(* Logix 5000 project; controller ARS14002_PLC vendor 1 type 14 code 218 rev 30.11; software revision 30.01 *)

TASK MainTask (continuous, watchdog 500 ms) : MainProgram
TASK PeriodicTask (periodic, rate 100 ms, priority 5, watchdog 1500 ms) : MainProgPeriodic

MODULES
   Local : vendor 1 type 14 code 218 (5069 0, rev 30.11)
      MAIN_PROCESSOR_T3_ENET : 1756-ENBT (Ethernet 192.168.23.100, rev 6.1, Output RPI 10 ms)   // PWHMI TOWER 3 ETHERNET MODULE
         MAIN_PROCESSOR_T3 : vendor 1 type 14 code 92 (ICP 0, rev 24.1, $d5a89411$ RPI 500 ms)   // PWHMI TOWER 3 PROCESSOR
      ARS14002_VFD800A : vendor 1 type 142 code 2192 (Ethernet 192.168.201.20, rev 13.3, Output RPI 20 ms)   // Cryo Pump 800A
          : vendor 1 type 142 code 16544 (RhinoBP 5, rev 1.1)
          : vendor 1 type 142 code 32928 (RhinoBP 13, rev 1.1)
          : vendor 1 type 142 code 767 (RhinoBP 2, rev 2.5)
          : vendor 1 type 142 code 57760 (RhinoBP 6, rev 1.2)
          : vendor 1 type 142 code 416 (RhinoBP 4, rev 1.8)
          : vendor 1 type 142 code 33184 (RhinoBP 14, rev 2.5)
      ARS14002_VFD800B : vendor 1 type 142 code 2192 (Ethernet 192.168.201.21, rev 13.3, Output RPI 20 ms)   // Cryo Pump 800B
          : vendor 1 type 142 code 416 (RhinoBP 4, rev 1.8)
          : vendor 1 type 142 code 767 (RhinoBP 2, rev 2.5)
          : vendor 1 type 142 code 32928 (RhinoBP 13, rev 1.1)
          : vendor 1 type 142 code 57760 (RhinoBP 6, rev 1.2)
          : vendor 1 type 142 code 33184 (RhinoBP 14, rev 2.5)
          : vendor 1 type 142 code 16544 (RhinoBP 5, rev 1.1)
      ARS14002_FVNR550 : vendor 1 type 3 code 506 (Ethernet 192.168.201.25, rev 5.1, Output RPI 20 ms)   // Vent Stack FAN-550
      ARS14002_FVR800C : vendor 1 type 3 code 548 (Ethernet 192.168.201.22, rev 5.1, Output RPI 20 ms)   // Cryo Pump 800C
      ARS14002_FVR800D : vendor 1 type 3 code 548 (Ethernet 192.168.201.23, rev 5.1, Output RPI 20 ms)   // Cryo Pump 800D
      MCP_S5 : 5069-IF8 (5069 5, rev 2.1, StandardDataDriven RPI 100 ms)
      MCP_S1 : 5069-IB16 (5069 1, rev 2.1, StandardDataDriven RPI 5 ms)
      MCP_S3 : vendor 1 type 7 code 1213 (5069 3, rev 3.1, StandardDataDriven RPI 5 ms)
      MCP_S4 : vendor 1 type 7 code 1213 (5069 4, rev 3.1, StandardDataDriven RPI 5 ms)
      MCP_S2 : vendor 1 type 7 code 1213 (5069 2, rev 3.1, StandardDataDriven RPI 5 ms)
      ARS14002_RCP1000 : 1734-AENTR (Ethernet 192.168.201.6, rev 5.1, Output RPI 20 ms)
         RCP1000_S13 : vendor 1 type 115 code 210 (PointIO 13, rev 3.1, Input RPI 80 ms)
         RCP1000_S1 : 1734-IB8 (PointIO 1, rev 3.1)
         RCP1000_S8 : vendor 1 type 115 code 49 (PointIO 8, rev 3.1, Input RPI 80 ms)
         RCP1000_S10 : vendor 1 type 115 code 49 (PointIO 10, rev 3.1, Input RPI 80 ms)
         RCP1000_S11 : vendor 1 type 115 code 49 (PointIO 11, rev 3.1, Input RPI 80 ms)
         RCP1000_S12 : vendor 1 type 115 code 210 (PointIO 12, rev 3.1, Input RPI 80 ms)
         RCP1000_S7 : vendor 1 type 115 code 49 (PointIO 7, rev 3.1, Input RPI 80 ms)
         RCP1000_S17 : vendor 1 type 115 code 49 (PointIO 17, rev 3.1, Input RPI 80 ms)
         RCP1000_S18 : vendor 1 type 115 code 49 (PointIO 18, rev 3.1, Input RPI 80 ms)
         RCP1000_S9 : vendor 1 type 115 code 49 (PointIO 9, rev 3.1, Input RPI 80 ms)
         RCP1000_S14 : vendor 1 type 115 code 210 (PointIO 14, rev 3.1, Input RPI 80 ms)
         RCP1000_S2 : 1734-IB8 (PointIO 2, rev 3.1)
         RCP1000_S3 : 1734-IB8 (PointIO 3, rev 3.1)
         RCP1000_S15 : vendor 1 type 115 code 211 (PointIO 15, rev 3.1, Output RPI 80 ms)
         RCP1000_S4 : 1734-OB8 (PointIO 4, rev 3.1)
         RCP1000_S6 : 1734-OB8 (PointIO 6, rev 3.1)
         RCP1000_S5 : 1734-OB8 (PointIO 5, rev 3.1)
         RCP1000_S16 : vendor 1 type 115 code 211 (PointIO 16, rev 3.1, Output RPI 80 ms)
      ARS14002_RCP600 : 1734-AENTR (Ethernet 192.168.201.4, rev 5.1, Output RPI 20 ms)
         RCP600_S7 : vendor 1 type 115 code 49 (PointIO 7, rev 3.1, Input RPI 80 ms)
         RCP600_S1 : 1734-IB8 (PointIO 1, rev 3.1)
         RCP600_S11 : vendor 1 type 115 code 210 (PointIO 11, rev 3.1, Input RPI 80 ms)
         RCP600_S9 : vendor 1 type 115 code 210 (PointIO 9, rev 3.1, Input RPI 80 ms)
         RCP600_S6 : vendor 1 type 115 code 49 (PointIO 6, rev 3.1, Input RPI 80 ms)
         RCP600_S10 : vendor 1 type 115 code 210 (PointIO 10, rev 3.1, Input RPI 80 ms)
         RCP600_S8 : vendor 1 type 115 code 49 (PointIO 8, rev 3.1, Input RPI 80 ms)
         RCP600_S5 : vendor 1 type 115 code 49 (PointIO 5, rev 3.1, Input RPI 80 ms)
         RCP600_S4 : 1734-OB8 (PointIO 4, rev 3.1)
         RCP600_S3 : 1734-OB8 (PointIO 3, rev 3.1)
         RCP600_S12 : vendor 1 type 115 code 211 (PointIO 12, rev 3.1, Output RPI 80 ms)
         RCP600_S13 : vendor 1 type 115 code 211 (PointIO 13, rev 3.1, Output RPI 80 ms)
         RCP600_S2 : 1734-OB8 (PointIO 2, rev 3.1)
      ARS14002_RCP800 : 1734-AENTR (Ethernet 192.168.201.5, rev 5.1, Output RPI 20 ms)
         RCP800_S23 : vendor 1 type 115 code 210 (PointIO 23, rev 3.1, Input RPI 80 ms)
         RCP800_S21 : vendor 1 type 115 code 210 (PointIO 21, rev 3.1, Input RPI 80 ms)
         RCP800_S17 : 1734-IR2 (PointIO 17, rev 3.1, Input RPI 80 ms)
         RCP800_S13 : 1734-IR2 (PointIO 13, rev 3.1, Input RPI 80 ms)
         RCP800_S2 : 1734-IB8 (PointIO 2, rev 3.1)
         RCP800_S16 : 1734-IR2 (PointIO 16, rev 3.1, Input RPI 80 ms)
         RCP800_S12 : vendor 1 type 115 code 49 (PointIO 12, rev 3.1, Input RPI 80 ms)
         RCP800_S22 : vendor 1 type 115 code 210 (PointIO 22, rev 3.1, Input RPI 80 ms)
         RCP800_S20 : 1734-IR2 (PointIO 20, rev 3.1, Input RPI 80 ms)
         RCP800_S24 : vendor 1 type 115 code 210 (PointIO 24, rev 3.1, Input RPI 80 ms)
         RCP800_S8 : 1734-IR2 (PointIO 8, rev 3.1, Input RPI 80 ms)
         RCP800_S11 : vendor 1 type 115 code 49 (PointIO 11, rev 3.1, Input RPI 80 ms)
         RCP800_S3 : 1734-IB8 (PointIO 3, rev 3.1)
         RCP800_S18 : 1734-IR2 (PointIO 18, rev 3.1, Input RPI 80 ms)
         RCP800_S14 : 1734-IR2 (PointIO 14, rev 3.1, Input RPI 80 ms)
         RCP800_S1 : 1734-IB8 (PointIO 1, rev 3.1)
         RCP800_S15 : 1734-IR2 (PointIO 15, rev 3.1, Input RPI 80 ms)
         RCP800_S10 : vendor 1 type 115 code 49 (PointIO 10, rev 3.1, Input RPI 80 ms)
         RCP800_S9 : 1734-IR2 (PointIO 9, rev 3.1, Input RPI 80 ms)
         RCP800_S19 : 1734-IR2 (PointIO 19, rev 3.1, Input RPI 80 ms)
         RCP800_S4 : 1734-OB8 (PointIO 4, rev 3.1)
         RCP800_S5 : 1734-OB8 (PointIO 5, rev 3.1)
         RCP800_S25 : vendor 1 type 115 code 211 (PointIO 25, rev 3.1, Output RPI 80 ms)
         RCP800_S7 : 1734-OB8 (PointIO 7, rev 3.1)
         RCP800_S6 : 1734-OB8 (PointIO 6, rev 3.1)
      ARS14002_RCP100 : 1734-AENTR (Ethernet 192.168.201.3, rev 5.1, Output RPI 20 ms)
         RCP100_S3 : vendor 1 type 115 code 49 (PointIO 3, rev 3.1, Input RPI 80 ms)
         RCP100_S5 : vendor 1 type 115 code 210 (PointIO 5, rev 3.1, Input RPI 80 ms)
         RCP100_S4 : vendor 1 type 115 code 49 (PointIO 4, rev 3.1, Input RPI 80 ms)
         RCP100_S6 : vendor 1 type 115 code 210 (PointIO 6, rev 3.1, Input RPI 80 ms)
         RCP100_S1 : 1734-IB8 (PointIO 1, rev 3.1)
         RCP100_S9 : 1734-OB8 (PointIO 9, rev 3.1)
         RCP100_S2 : 1734-OB8 (PointIO 2, rev 3.1)
         RCP100_S7 : vendor 1 type 115 code 211 (PointIO 7, rev 3.1, Output RPI 80 ms)
         RCP100_S8 : vendor 1 type 115 code 211 (PointIO 8, rev 3.1, Output RPI 80 ms)
END_MODULES

TYPE UDT_IPC :
STRUCT
   ConnectionStatus : CONNECTION_STATUS;
   BOOL : BOOL[32];
   REAL : REAL[32];
   DINT : DINT[32];
END_STRUCT
END_TYPE

ADD_ON_INSTRUCTION CM_AI_SCL   (* revision 2.0, vendor EVERWORKS *)
// Analog Input
VAR_INPUT
   RawMin : INT := 4000; {required}   // Config Raw Min
   RawMax : INT := 20000; {required}   // Config Raw Max
   EuMin : REAL; {visible}   // Config Min EU
   EuMax : REAL := 100.0; {visible}   // Config Max EU
   In_Raw : INT; {required}   // Channel Raw Count
END_VAR
VAR_OUTPUT
   Percent : REAL; {access Read Only}   // Scaled % of PV
   PV : REAL; {access Read Only, visible}   // Scaled PV
END_VAR

ROUTINE Logic   (* ladder *)
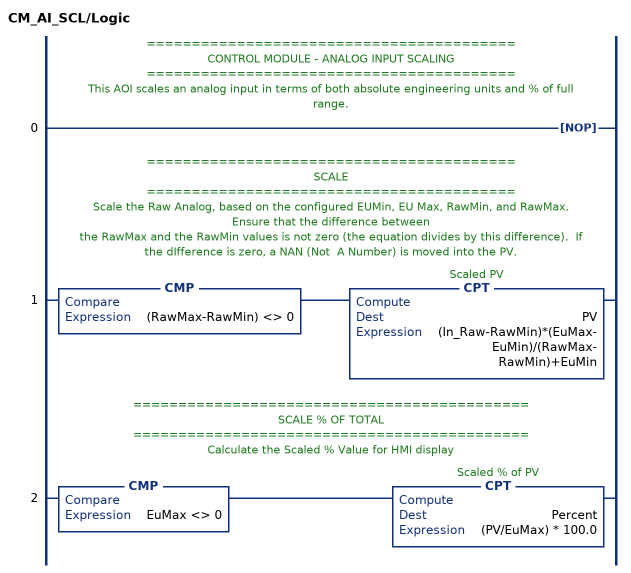
   // =========================================
   // CONTROL MODULE - ANALOG INPUT SCALING
   // =========================================
   // This AOI scales an analog input in terms of both absolute engineering units and % of full range.
   0: NOP();
   // =========================================
   // SCALE
   // =========================================
   // Scale the Raw Analog, based on the configured EUMin, EU Max, RawMin, and RawMax.  Ensure that the difference between
   // the RawMax and the RawMin values is not zero (the equation divides by this difference).  If the dIfference is zero, a NAN (Not  A Number) is moved into the PV.
   1: CMP((RawMax-RawMin) <> 0)CPT(PV,(In_Raw-RawMin)*(EuMax-EuMin)/(RawMax-RawMin)+EuMin);
   // ============================================
   // SCALE % OF TOTAL
   // ============================================
   // Calculate the Scaled % Value for HMI display
   2: CMP(EuMax <> 0)CPT(Percent,(PV/EuMax) * 100.0);
END_ROUTINE
END_ADD_ON_INSTRUCTION

ADD_ON_INSTRUCTION CM_AI_SCL_ALT   (* revision 2.0, vendor EVERWORKS *)
// Analog Input with Alt Scaling
VAR_INPUT
   RawMin : INT := 4000; {required}   // Config Raw Min
   RawMax : INT := 20000; {required}   // Config Raw Max
   EuMin : REAL; {visible}   // Config Min EU
   EuMax : REAL := 100.0; {visible}   // Config Max EU
   AltScaleMultiplier : REAL; {required}   // Alternate Scale Multiplier
   In_Raw : INT; {required}   // Channel Raw Count
END_VAR
VAR_OUTPUT
   Percent : REAL; {access Read Only}   // Scaled % of PV
   PV : REAL; {access Read Only, visible}   // Scaled PV
   AltScalePV : REAL; {visible}   // Alternate Scaled PV
END_VAR

ROUTINE Logic   (* ladder *)
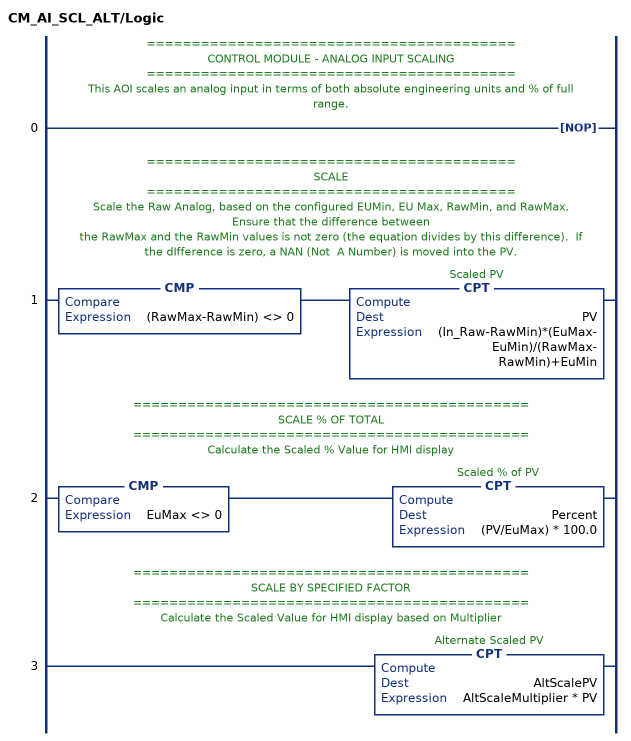
   // =========================================
   // CONTROL MODULE - ANALOG INPUT SCALING
   // =========================================
   // This AOI scales an analog input in terms of both absolute engineering units and % of full range.
   0: NOP();
   // =========================================
   // SCALE
   // =========================================
   // Scale the Raw Analog, based on the configured EUMin, EU Max, RawMin, and RawMax.  Ensure that the difference between
   // the RawMax and the RawMin values is not zero (the equation divides by this difference).  If the dIfference is zero, a NAN (Not  A Number) is moved into the PV.
   1: CMP((RawMax-RawMin) <> 0)CPT(PV,(In_Raw-RawMin)*(EuMax-EuMin)/(RawMax-RawMin)+EuMin);
   // ============================================
   // SCALE % OF TOTAL
   // ============================================
   // Calculate the Scaled % Value for HMI display
   2: CMP(EuMax <> 0)CPT(Percent,(PV/EuMax) * 100.0);
   // ============================================
   // SCALE BY SPECIFIED FACTOR
   // ============================================
   // Calculate the Scaled Value for HMI display based on Multiplier
   3: CPT(AltScalePV,AltScaleMultiplier * PV);
END_ROUTINE
END_ADD_ON_INSTRUCTION

ADD_ON_INSTRUCTION CM_AO_SCL   (* revision 2.0, vendor EVERWORKS *)
// Analog Output
VAR_OUTPUT
   EngValue : REAL; {access Read Only, visible}   // Scaled Engineering Value
   Percent : REAL; {access Read Only}   // Scaled % of PV
   Out_Raw : INT; {required}   // Channel Raw Count
END_VAR
VAR_INPUT
   EuMin : REAL; {visible}   // Config Min EU
   EuMax : REAL := 100.0; {visible}   // Config Max EU
   RawMin : INT := 4000; {required}   // Config Raw Min
   RawMax : INT := 20000; {required}   // Config Raw Max
END_VAR

ROUTINE Logic   (* ladder *)
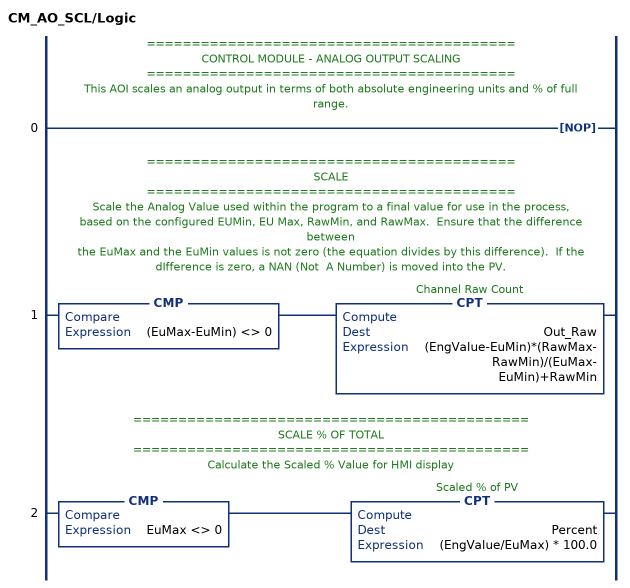
   // =========================================
   // CONTROL MODULE - ANALOG OUTPUT SCALING
   // =========================================
   // This AOI scales an analog output in terms of both absolute engineering units and % of full range.
   0: NOP();
   // =========================================
   // SCALE
   // =========================================
   // Scale the Analog Value used within the program to a final value for use in the process, based on the configured EUMin, EU Max, RawMin, and RawMax.  Ensure that the difference between
   // the EuMax and the EuMin values is not zero (the equation divides by this difference).  If the dIfference is zero, a NAN (Not  A Number) is moved into the PV.
   1: CMP((EuMax-EuMin) <> 0)CPT(Out_Raw,(EngValue-EuMin)*(RawMax-RawMin)/(EuMax-EuMin)+RawMin);
   // ============================================
   // SCALE % OF TOTAL
   // ============================================
   // Calculate the Scaled % Value for HMI display
   2: CMP(EuMax <> 0)CPT(Percent,(EngValue/EuMax) * 100.0);
END_ROUTINE
END_ADD_ON_INSTRUCTION

ADD_ON_INSTRUCTION CM_AO_VLV   (* revision 2.0, vendor EVERWORKS *)
// Modulating Valve
VAR_INPUT
   FailPos : BOOL; {required}   // Fail Position (0=Fail Closed, 1=Fail Open)
   EuMin : REAL; {visible}   // Config Min EU
   EuMax : REAL := 100.0; {visible}   // Config Max EU
   RawMin : INT := 4000; {required}   // Config Raw Min
   RawMax : INT := 20000; {required}   // Config Raw Max
   ZT : REAL; {required}   // Position Feedback (EU)
   EngValue : REAL; {access Read Only, visible}   // Scaled Engineering Value
END_VAR
VAR_OUTPUT
   Out_Raw : INT; {required}   // Channel Raw Count
   Alm_Dev : BOOL; {visible}   // Deviation Alarm
END_VAR
VAR_INPUT
   Alm_Dev_SP : REAL := 10.0;   // % Deviation between CV and ZT allowed
   Alm_Dev_TmrPre : DINT := 5;   // Deviation Alarm Delay Timer Preset (seconds)
END_VAR
VAR
   Alm_Dev_Tmr : TIMER := (PRE := 5000); {access None}   // Deviation Alarm Delay Timer
   Comp_Overshoot : REAL; {access None}   // ZT (position feedback) - CV (commanded position)
   Comp_Undershoot : REAL; {access None}   // CV (commanded position) - ZT (position feedback)
END_VAR

ROUTINE Logic   (* ladder *)
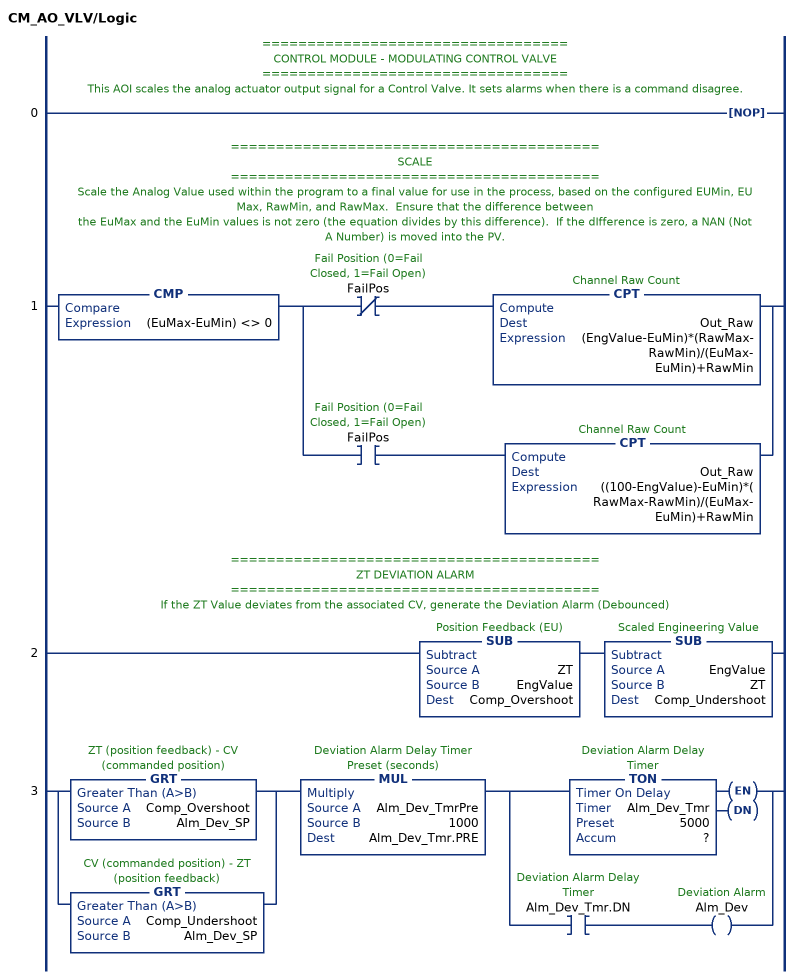
   // ==================================
   // CONTROL MODULE - MODULATING CONTROL VALVE
   // ==================================
   // This AOI scales the analog actuator output signal for a Control Valve. It sets alarms when there is a command disagree.
   0: NOP();
   // =========================================
   // SCALE
   // =========================================
   // Scale the Analog Value used within the program to a final value for use in the process, based on the configured EUMin, EU Max, RawMin, and RawMax.  Ensure that the difference between
   // the EuMax and the EuMin values is not zero (the equation divides by this difference).  If the dIfference is zero, a NAN (Not  A Number) is moved into the PV.
   1: CMP((EuMax-EuMin) <> 0)[XIO(FailPos) CPT(Out_Raw,(EngValue-EuMin)*(RawMax-RawMin)/(EuMax-EuMin)+RawMin) ,XIC(FailPos) CPT(Out_Raw,((100-EngValue)-EuMin)*(RawMax-RawMin)/(EuMax-EuMin)+RawMin) ];
   // =========================================
   // ZT DEVIATION ALARM
   // =========================================
   // If the ZT Value deviates from the associated CV, generate the Deviation Alarm (Debounced)
   2: SUB(ZT,EngValue,Comp_Overshoot)SUB(EngValue,ZT,Comp_Undershoot);
   3: [GRT(Comp_Overshoot,Alm_Dev_SP) ,GRT(Comp_Undershoot,Alm_Dev_SP) ]MUL(Alm_Dev_TmrPre,1000,Alm_Dev_Tmr.PRE)[TON(Alm_Dev_Tmr,?,?) ,XIC(Alm_Dev_Tmr.DN) OTE(Alm_Dev) ];
END_ROUTINE
END_ADD_ON_INSTRUCTION

ADD_ON_INSTRUCTION CM_DO_FVNR   (* revision 2.0, vendor EVERWORKS *)
// FVNR Starter
VAR_INPUT
   ILW : DINT;   // InterLocks Word
   Auto : BOOL; {visible}   // Starter Mode (0=Manual, 1=Auto)
   AlmCurrentLow_SP : REAL; {visible}   // Low Current Setpoint
   AlmCurrentHigh_SP : REAL := 999.0; {visible}   // High Current Setpoint
   Current : REAL; {access Read Only, visible}   // Motor Current Feedback
   Flt : BOOL; {visible}   // Fault Status
   AlmCD_TmrPre : DINT := 5;   // Command Disagree Alarm Delay Timer Preset (Seconds)
END_VAR
VAR_OUTPUT
   Intlk : BOOL; {access Read Only, visible}   // Interlocked Status
END_VAR
VAR_INPUT
   ProgStartReq : BOOL;   // Program Start Request
END_VAR
VAR_OUTPUT
   AlmCD : BOOL; {access Read Only, visible}   // Command Disagree Alarm
END_VAR
VAR_INPUT
   Running : BOOL; {visible}   // Motor Running Status
END_VAR
VAR_OUTPUT
   Out : BOOL; {required}   // Start Command
   AlmCurrentLow : BOOL; {visible}   // Low Current Alarm
   AlmCurrentHigh : BOOL; {visible}   // High Current Alarm
END_VAR
VAR_INPUT
   AlmCurrent_TmrPre : DINT := 5;   // Low Current Alarm Delay Timer Preset (Seconds)
   OperStartReq : BOOL;   // Manual Start Request
END_VAR
VAR
   AlmCD_Tmr : TIMER := (PRE := 5000); {access None}   // Command Disagree Alarm Delay Timer
   ILW_Desc : STRING[14];
   AlmCurrentLow_Tmr : TIMER := (PRE := 5000); {access None}   // Low Current Alarm Delay Timer
   AutoManTransOSR_SB : BOOL; {access None}
   AutoManTransOSR_OB : BOOL; {access None}
   AlmCurrentHigh_Tmr : TIMER := (PRE := 5000); {access None}   // High Current Alarm Delay Timer
END_VAR

ROUTINE Logic   (* ladder *)
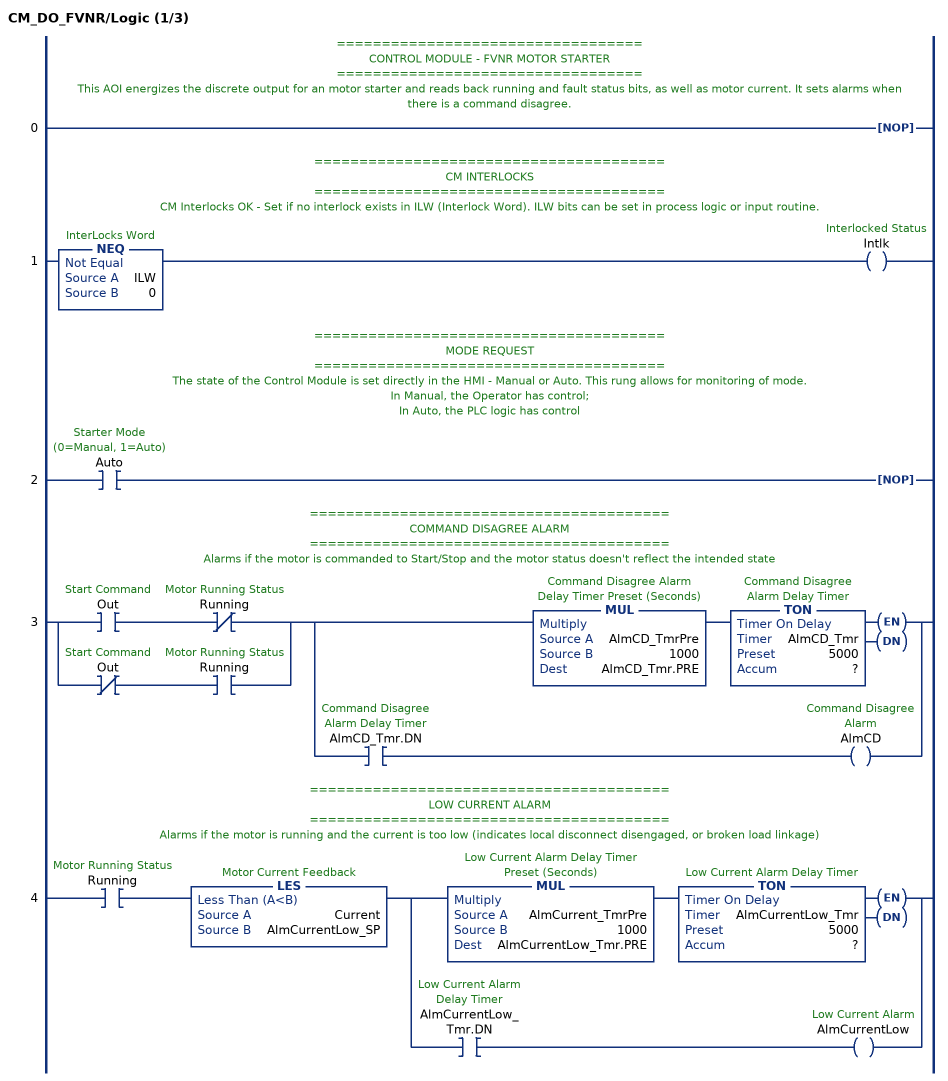
   // ==================================
   // CONTROL MODULE - FVNR MOTOR STARTER
   // ==================================
   // This AOI energizes the discrete output for an motor starter and reads back running and fault status bits, as well as motor current. It sets alarms when there is a command disagree.
   0: NOP();
   // =======================================
   // CM INTERLOCKS
   // =======================================
   // CM Interlocks OK - Set if no interlock exists in ILW (Interlock Word). ILW bits can be set in process logic or input routine.
   1: NEQ(ILW,0)OTE(Intlk);
   // =======================================
   // MODE REQUEST
   // =======================================
   // The state of the Control Module is set directly in the HMI - Manual or Auto. This rung allows for monitoring of mode.
   // In Manual, the Operator has control;
   //  In Auto, the PLC logic has control
   2: XIC(Auto)NOP();
   // ========================================
   // COMMAND DISAGREE ALARM
   // ========================================
   // Alarms if the motor is commanded to Start/Stop and the motor status doesn't reflect the intended state
   3: [XIC(Out) XIO(Running) ,XIO(Out) XIC(Running) ][MUL(AlmCD_TmrPre,1000,AlmCD_Tmr.PRE) TON(AlmCD_Tmr,?,?) ,XIC(AlmCD_Tmr.DN) OTE(AlmCD) ];
   // ========================================
   // LOW CURRENT ALARM
   // ========================================
   // Alarms if the motor is running and the current is too low (indicates local disconnect disengaged, or broken load linkage)
   4: XIC(Running)LES(Current,AlmCurrentLow_SP)[MUL(AlmCurrent_TmrPre,1000,AlmCurrentLow_Tmr.PRE) TON(AlmCurrentLow_Tmr,?,?) ,XIC(AlmCurrentLow_Tmr.DN) OTE(AlmCurrentLow) ];
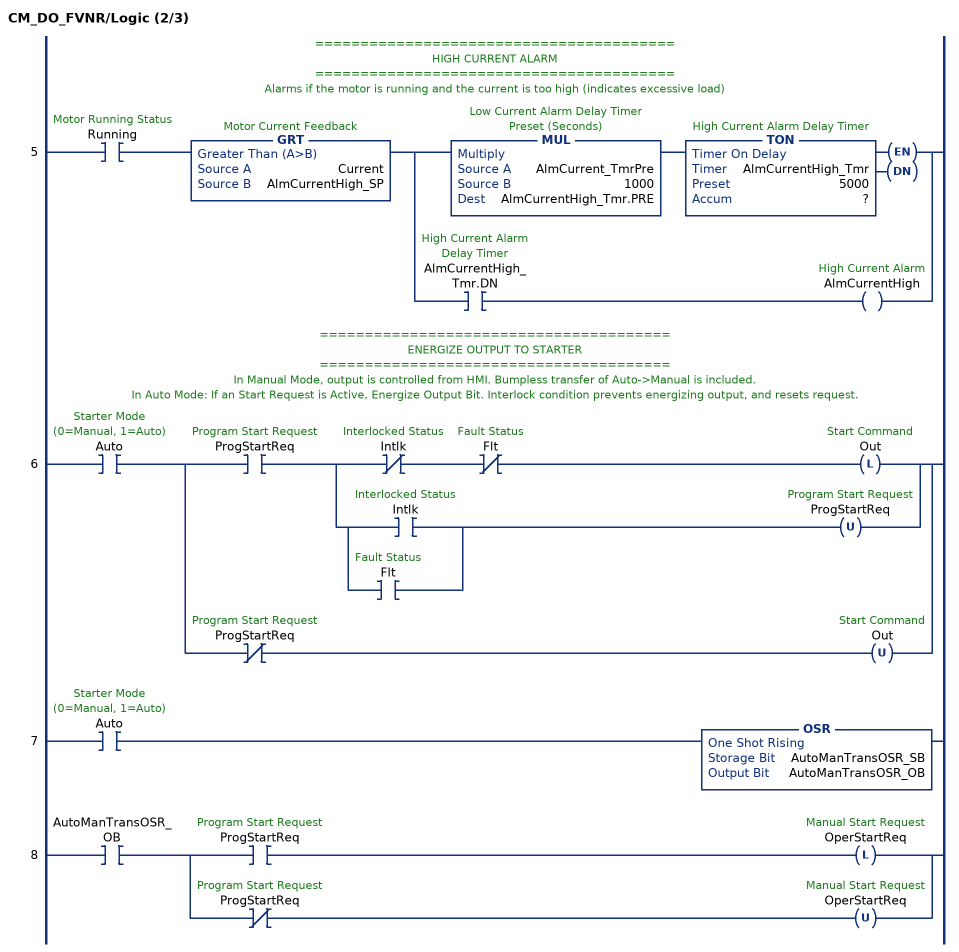
   // ========================================
   // HIGH CURRENT ALARM
   // ========================================
   // Alarms if the motor is running and the current is too high (indicates excessive load)
   5: XIC(Running)GRT(Current,AlmCurrentHigh_SP)[MUL(AlmCurrent_TmrPre,1000,AlmCurrentHigh_Tmr.PRE) TON(AlmCurrentHigh_Tmr,?,?) ,XIC(AlmCurrentHigh_Tmr.DN) OTE(AlmCurrentHigh) ];
   // =======================================
   // ENERGIZE OUTPUT TO STARTER
   // =======================================
   // In Manual Mode, output is controlled from HMI. Bumpless transfer of Auto->Manual is included.
   // In Auto Mode: If an Start Request is Active, Energize Output Bit. Interlock condition prevents energizing output, and resets request.
   6: XIC(Auto)[XIC(ProgStartReq) [XIO(Intlk) XIO(Flt) OTL(Out) ,[XIC(Intlk) ,XIC(Flt) ] OTU(ProgStartReq) ] ,XIO(ProgStartReq) OTU(Out) ];
   7: XIC(Auto)OSR(AutoManTransOSR_SB,AutoManTransOSR_OB);
   8: XIC(AutoManTransOSR_OB)[XIC(ProgStartReq) OTL(OperStartReq) ,XIO(ProgStartReq) OTU(OperStartReq) ];
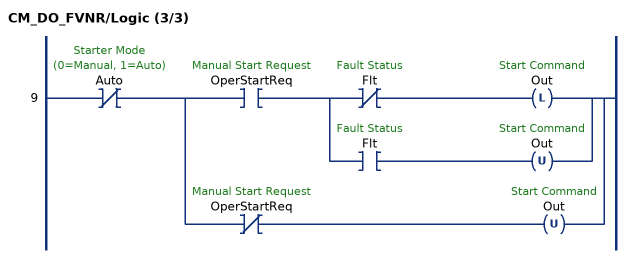
   9: XIO(Auto)[XIC(OperStartReq) [XIO(Flt) OTL(Out) ,XIC(Flt) OTU(Out) ] ,XIO(OperStartReq) OTU(Out) ];
END_ROUTINE
END_ADD_ON_INSTRUCTION

ADD_ON_INSTRUCTION CM_DO_FVR   (* revision 2.0, vendor EVERWORKS *)
// FVR Starter
VAR_INPUT
   ILW : DINT;   // InterLocks Word
   Auto : BOOL; {visible}   // Starter Mode (0=Manual, 1=Auto)
   AlmCurrentLow_SP : REAL; {visible}   // Low Current Setpoint
   AlmCurrentHigh_SP : REAL := 999.0; {visible}   // High Current Setpoint
   Current : REAL; {access Read Only, visible}   // Motor Current Feedback
   Flt : BOOL; {visible}   // Fault Status
   AlmCD_TmrPre : DINT := 5;   // Command Disagree Alarm Delay Timer Preset (Seconds)
END_VAR
VAR_OUTPUT
   Intlk : BOOL; {access Read Only, visible}   // Interlocked Status
END_VAR
VAR_INPUT
   ProgStartReq : BOOL;   // Program Start Request
END_VAR
VAR_OUTPUT
   AlmCD : BOOL; {access Read Only, visible}   // Command Disagree Alarm
END_VAR
VAR_INPUT
   Direction : BOOL; {visible}   // Motor Direction 0=Forward 1=Reverse
   RunningFwd : BOOL; {visible}   // Motor Running Forward Status
   RunningRvs : BOOL; {visible}   // Motor Running Reverse Status
END_VAR
VAR_OUTPUT
   OutFwd : BOOL; {required}   // Start Command Forward
   OutRvs : BOOL; {access Read Only, required}   // Start Command Reverse
   AlmCurrentLow : BOOL; {visible}   // Low Current Alarm
   AlmCurrentHigh : BOOL; {visible}   // High Current Alarm
END_VAR
VAR_INPUT
   AlmCurrent_TmrPre : DINT := 5;   // Low Current Alarm Delay Timer Preset (Seconds)
   OperStartReq : BOOL;   // Manual Start Request
END_VAR
VAR
   AlmCD_Tmr : TIMER := (PRE := 5000); {access None}   // Command Disagree Alarm Delay Timer
   ILW_Desc : STRING[14];
   AlmCurrentLow_Tmr : TIMER := (PRE := 5000); {access None}   // Low Current Alarm Delay Timer
   AutoManTransOSR_SB : BOOL; {access None}
   AutoManTransOSR_OB : BOOL; {access None}
   AlmCurrentHigh_Tmr : TIMER := (PRE := 5000); {access None}   // High Current Alarm Delay Timer
END_VAR

ROUTINE Logic   (* ladder *)
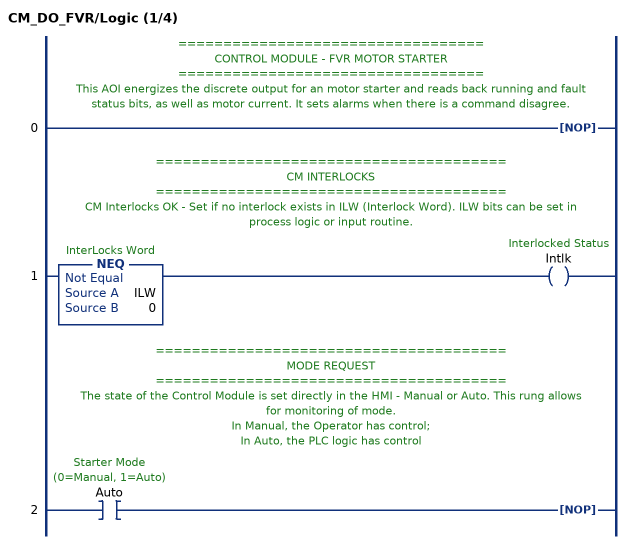
   // ==================================
   // CONTROL MODULE - FVR MOTOR STARTER
   // ==================================
   // This AOI energizes the discrete output for an motor starter and reads back running and fault status bits, as well as motor current. It sets alarms when there is a command disagree.
   0: NOP();
   // =======================================
   // CM INTERLOCKS
   // =======================================
   // CM Interlocks OK - Set if no interlock exists in ILW (Interlock Word). ILW bits can be set in process logic or input routine.
   1: NEQ(ILW,0)OTE(Intlk);
   // =======================================
   // MODE REQUEST
   // =======================================
   // The state of the Control Module is set directly in the HMI - Manual or Auto. This rung allows for monitoring of mode.
   // In Manual, the Operator has control;
   //  In Auto, the PLC logic has control
   2: XIC(Auto)NOP();
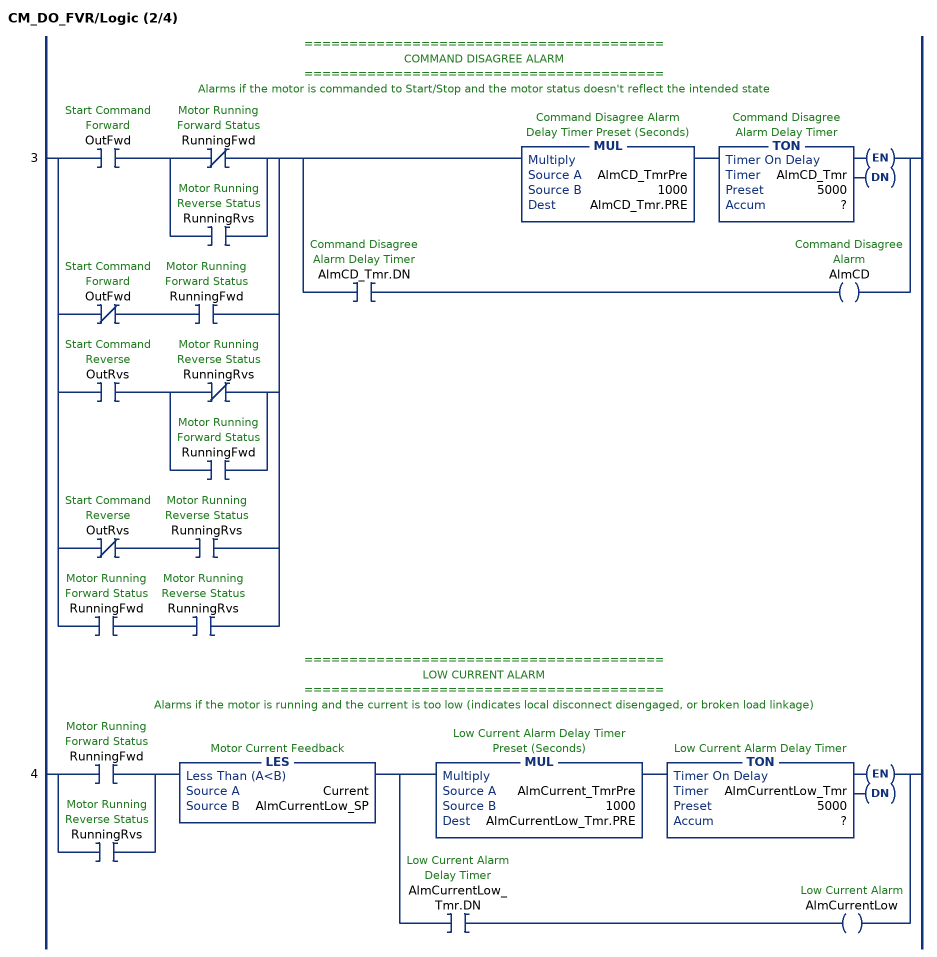
   // ========================================
   // COMMAND DISAGREE ALARM
   // ========================================
   // Alarms if the motor is commanded to Start/Stop and the motor status doesn't reflect the intended state
   3: [XIC(OutFwd) [XIO(RunningFwd) ,XIC(RunningRvs) ] ,XIO(OutFwd) XIC(RunningFwd) ,XIC(OutRvs) [XIO(RunningRvs) ,XIC(RunningFwd) ] ,XIO(OutRvs) XIC(RunningRvs) ,XIC(RunningFwd) XIC(RunningRvs) ][MUL(AlmCD_TmrPre,1000,AlmCD_Tmr.PRE) TON(AlmCD_Tmr,?,?) ,XIC(AlmCD_Tmr.DN) OTE(AlmCD) ];
   // ========================================
   // LOW CURRENT ALARM
   // ========================================
   // Alarms if the motor is running and the current is too low (indicates local disconnect disengaged, or broken load linkage)
   4: [XIC(RunningFwd) ,XIC(RunningRvs) ]LES(Current,AlmCurrentLow_SP)[MUL(AlmCurrent_TmrPre,1000,AlmCurrentLow_Tmr.PRE) TON(AlmCurrentLow_Tmr,?,?) ,XIC(AlmCurrentLow_Tmr.DN) OTE(AlmCurrentLow) ];
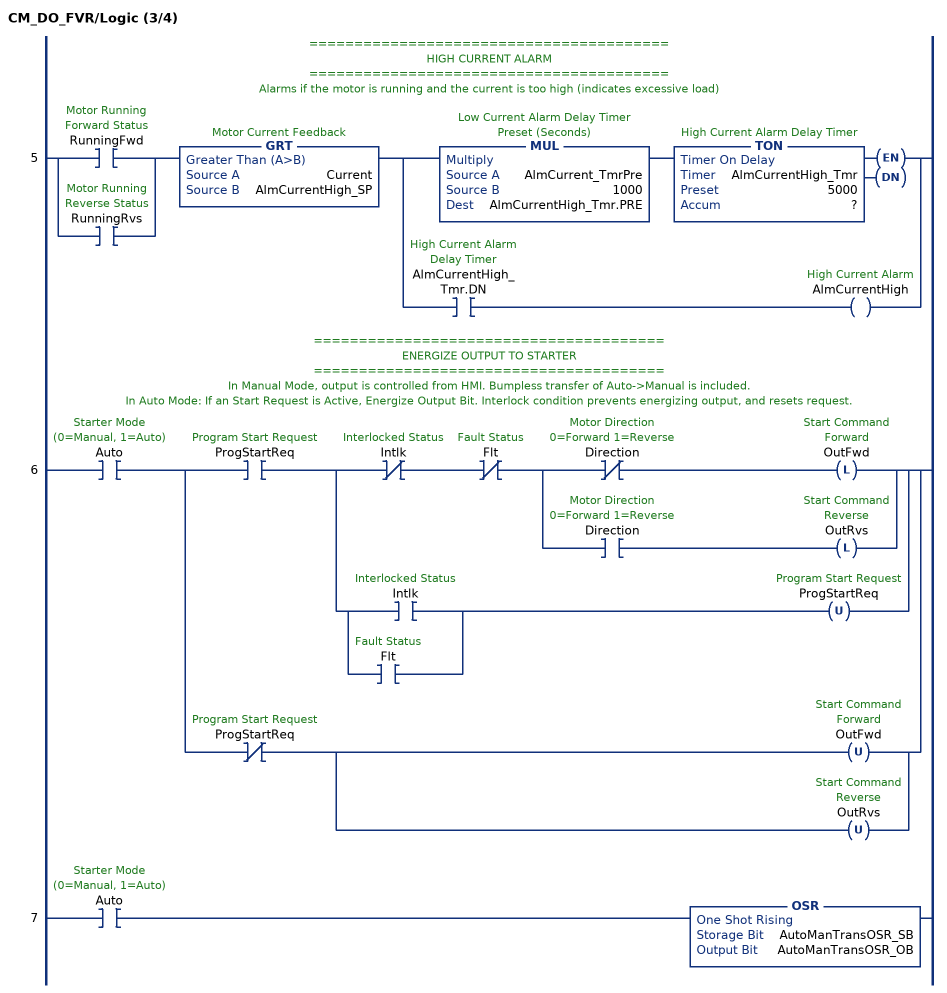
   // ========================================
   // HIGH CURRENT ALARM
   // ========================================
   // Alarms if the motor is running and the current is too high (indicates excessive load)
   5: [XIC(RunningFwd) ,XIC(RunningRvs) ]GRT(Current,AlmCurrentHigh_SP)[MUL(AlmCurrent_TmrPre,1000,AlmCurrentHigh_Tmr.PRE) TON(AlmCurrentHigh_Tmr,?,?) ,XIC(AlmCurrentHigh_Tmr.DN) OTE(AlmCurrentHigh) ];
   // =======================================
   // ENERGIZE OUTPUT TO STARTER
   // =======================================
   // In Manual Mode, output is controlled from HMI. Bumpless transfer of Auto->Manual is included.
   // In Auto Mode: If an Start Request is Active, Energize Output Bit. Interlock condition prevents energizing output, and resets request.
   6: XIC(Auto)[XIC(ProgStartReq) [XIO(Intlk) XIO(Flt) [XIO(Direction) OTL(OutFwd) ,XIC(Direction) OTL(OutRvs) ] ,[XIC(Intlk) ,XIC(Flt) ] OTU(ProgStartReq) ] ,XIO(ProgStartReq) [OTU(OutFwd) ,OTU(OutRvs) ] ];
   7: XIC(Auto)OSR(AutoManTransOSR_SB,AutoManTransOSR_OB);
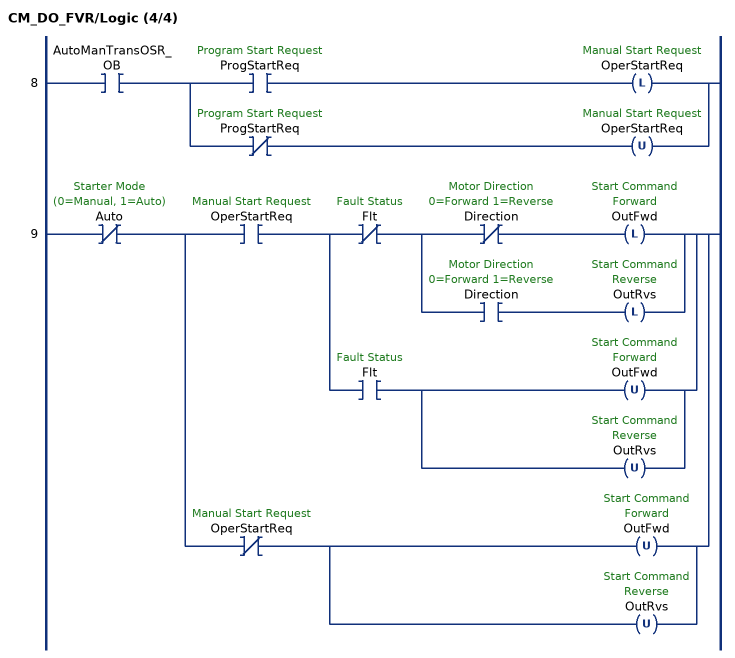
   8: XIC(AutoManTransOSR_OB)[XIC(ProgStartReq) OTL(OperStartReq) ,XIO(ProgStartReq) OTU(OperStartReq) ];
   9: XIO(Auto)[XIC(OperStartReq) [XIO(Flt) [XIO(Direction) OTL(OutFwd) ,XIC(Direction) OTL(OutRvs) ] ,XIC(Flt) [OTU(OutFwd) ,OTU(OutRvs) ] ] ,XIO(OperStartReq) [OTU(OutFwd) ,OTU(OutRvs) ] ];
END_ROUTINE
END_ADD_ON_INSTRUCTION

ADD_ON_INSTRUCTION CM_DO_GENERIC   (* revision 2.0, vendor EVERWORKS *)
// On/Off Device (No Feedback)
VAR_INPUT
   ILW : DINT;   // InterLocks Word
   FailPos : BOOL; {visible}   // Fail Position (0=Fail Closed, 1=Fail Open)
   Auto : BOOL; {visible}   // Device Mode (0=Manual, 1=Auto)
END_VAR
VAR_OUTPUT
   Intlk : BOOL; {access Read Only, visible}   // Interlocked Status
END_VAR
VAR_INPUT
   EnergizeReq : BOOL; {visible}   // Program Energize Request
END_VAR
VAR_OUTPUT
   Out : BOOL; {required}   // Energize Command
END_VAR
VAR_INPUT
   DeenergizeONS : BOOL;   // Bit Reserved for De-energize ONS
END_VAR
VAR
   ILW_Desc : STRING[14];
END_VAR

ROUTINE Logic   (* ladder *)
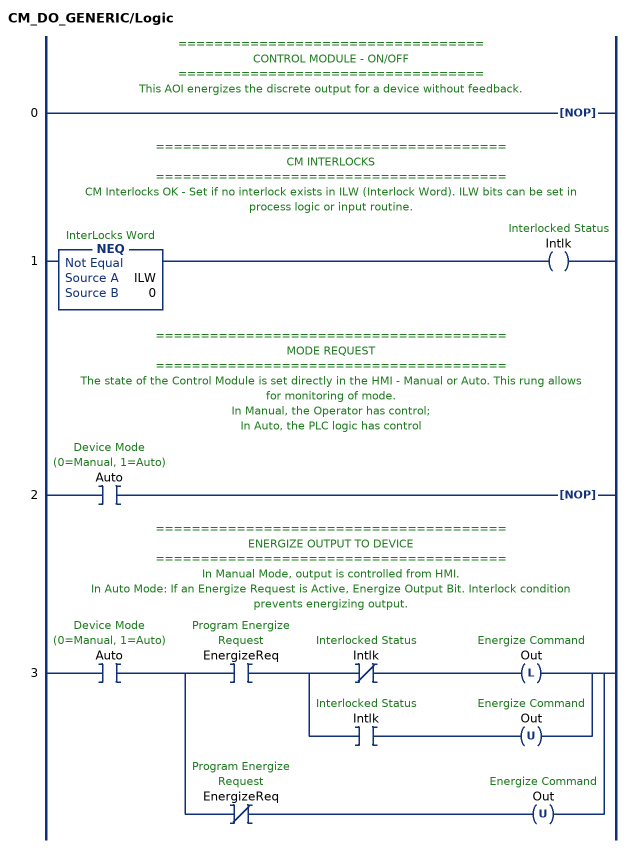
   // ==================================
   // CONTROL MODULE - ON/OFF
   // ==================================
   // This AOI energizes the discrete output for a device without feedback.
   0: NOP();
   // =======================================
   // CM INTERLOCKS
   // =======================================
   // CM Interlocks OK - Set if no interlock exists in ILW (Interlock Word). ILW bits can be set in process logic or input routine.
   1: NEQ(ILW,0)OTE(Intlk);
   // =======================================
   // MODE REQUEST
   // =======================================
   // The state of the Control Module is set directly in the HMI - Manual or Auto. This rung allows for monitoring of mode.
   // In Manual, the Operator has control;
   //  In Auto, the PLC logic has control
   2: XIC(Auto)NOP();
   // =======================================
   // ENERGIZE OUTPUT TO DEVICE
   // =======================================
   // In Manual Mode, output is controlled from HMI.
   // In Auto Mode: If an Energize Request is Active, Energize Output Bit. Interlock condition prevents energizing output.
   3: XIC(Auto)[XIC(EnergizeReq) [XIO(Intlk) OTL(Out) ,XIC(Intlk) OTU(Out) ] ,XIO(EnergizeReq) OTU(Out) ];
END_ROUTINE
END_ADD_ON_INSTRUCTION

ADD_ON_INSTRUCTION CM_DO_VLV   (* revision 2.0, vendor EVERWORKS *)
// On/Off Valve
VAR_INPUT
   FailPos : BOOL; {access Read Only, required}   // Valve Fail Position (0=Fail Closed, 1=Fail Open)
   ILW : DINT;   // InterLocks Word
   Auto : BOOL; {visible}   // Valve Mode (0=Manual, 1=Auto)
   Open : BOOL; {visible}   // Valve Open Status
   Closed : BOOL; {visible}   // Valve Closed Status
   AlmCD_TmrPre : DINT := 5;   // Command Disagree Alarm Delay Timer Preset (Seconds)
END_VAR
VAR_OUTPUT
   Intlk : BOOL; {access Read Only, visible}   // Interlocked Status
END_VAR
VAR_INPUT
   EnergizeReq : BOOL; {visible}   // Program Valve Open Request
END_VAR
VAR_OUTPUT
   AlmCD : BOOL; {access Read Only, visible}   // Command Disagree Alarm
   Transition : BOOL; {access Read Only}   // Valve in Transition
   Out : BOOL; {required}   // Valve Open Command
END_VAR
VAR_INPUT
   DeenergizeONS : BOOL;   // Bit Reserved for De-energize ONS
END_VAR
VAR
   AlmCD_Tmr : TIMER := (PRE := 5000); {access None}   // Command Disagree Alarm Delay Timer
   ILW_Desc : STRING[14];
END_VAR

ROUTINE Logic   (* ladder *)
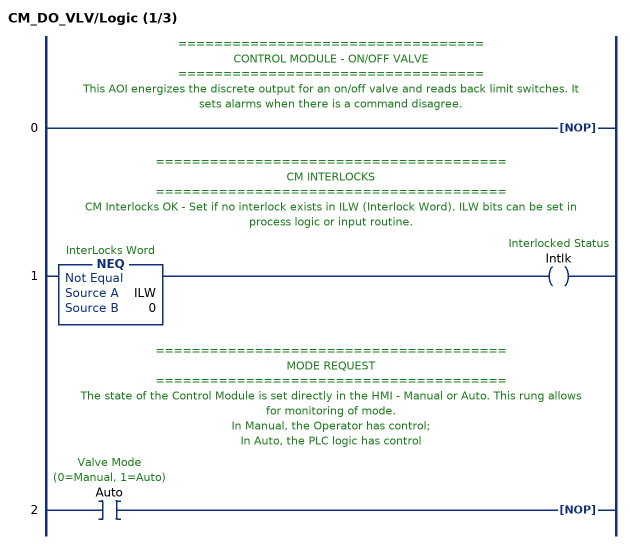
   // ==================================
   // CONTROL MODULE - ON/OFF VALVE
   // ==================================
   // This AOI energizes the discrete output for an on/off valve and reads back limit switches. It sets alarms when there is a command disagree.
   0: NOP();
   // =======================================
   // CM INTERLOCKS
   // =======================================
   // CM Interlocks OK - Set if no interlock exists in ILW (Interlock Word). ILW bits can be set in process logic or input routine.
   1: NEQ(ILW,0)OTE(Intlk);
   // =======================================
   // MODE REQUEST
   // =======================================
   // The state of the Control Module is set directly in the HMI - Manual or Auto. This rung allows for monitoring of mode.
   // In Manual, the Operator has control;
   //  In Auto, the PLC logic has control
   2: XIC(Auto)NOP();
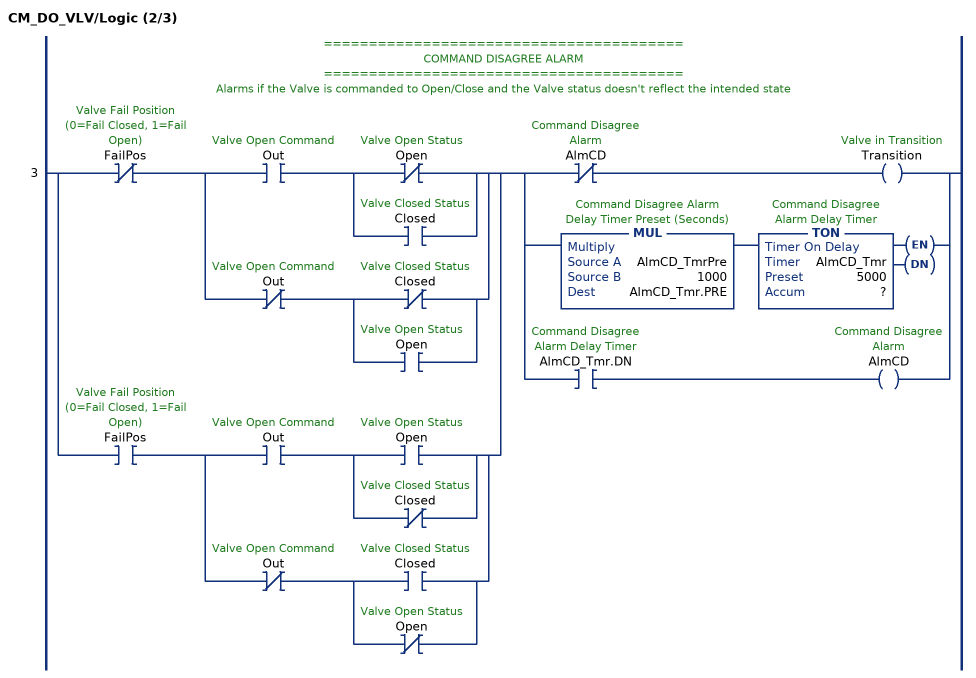
   // ========================================
   // COMMAND DISAGREE ALARM
   // ========================================
   // Alarms if the Valve is commanded to Open/Close and the Valve status doesn't reflect the intended state
   3: [XIO(FailPos) [XIC(Out) [XIO(Open) ,XIC(Closed) ] ,XIO(Out) [XIO(Closed) ,XIC(Open) ] ] ,XIC(FailPos) [XIC(Out) [XIC(Open) ,XIO(Closed) ] ,XIO(Out) [XIC(Closed) ,XIO(Open) ] ] ][XIO(AlmCD) OTE(Transition) ,MUL(AlmCD_TmrPre,1000,AlmCD_Tmr.PRE) TON(AlmCD_Tmr,?,?) ,XIC(AlmCD_Tmr.DN) OTE(AlmCD) ];
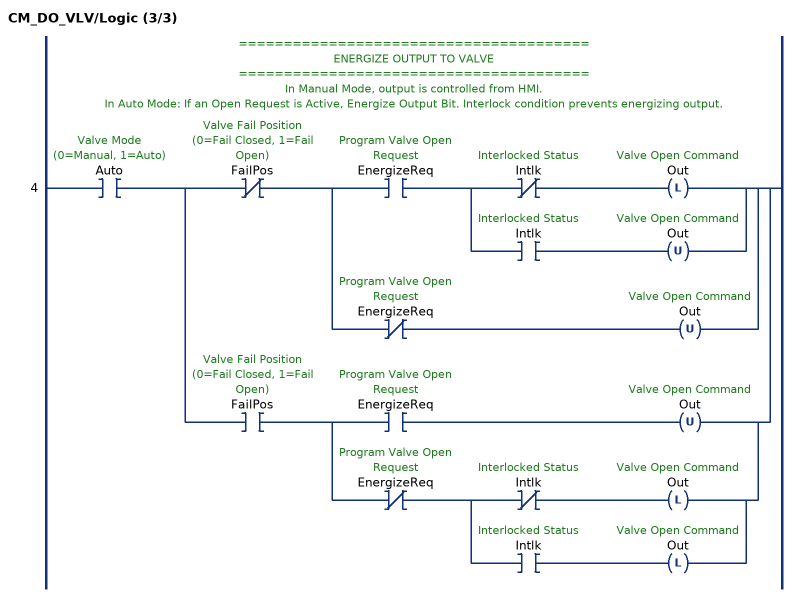
   // =======================================
   // ENERGIZE OUTPUT TO VALVE
   // =======================================
   // In Manual Mode, output is controlled from HMI.
   // In Auto Mode: If an Open Request is Active, Energize Output Bit. Interlock condition prevents energizing output.
   4: XIC(Auto)[XIO(FailPos) [XIC(EnergizeReq) [XIO(Intlk) OTL(Out) ,XIC(Intlk) OTU(Out) ] ,XIO(EnergizeReq) OTU(Out) ] ,XIC(FailPos) [XIC(EnergizeReq) OTU(Out) ,XIO(EnergizeReq) [XIO(Intlk) OTL(Out) ,XIC(Intlk) OTL(Out) ] ] ];
END_ROUTINE
END_ADD_ON_INSTRUCTION

VAR_GLOBAL   (* controller tags *)
   AC_OK_1000 : BOOL := 1;
   AC_OK_600 : BOOL := 1;
   AC_OK_800 : BOOL := 1;
   AC_OK_MCP : BOOL := 1;
   AN_1000_HI_PPM_SHUTDOWN : BOOL;   // **future use
   AN_1000A : CM_AI_SCL := (RawMax := 10000, EuMax := 1000.0, In_Raw := 122, Percent := 1.22, PV := 12.2);
   AN_1000A_RESTART_TMR : TIMER := (PRE := 10000);
   AN_1000A_SP : REAL := 50.0;
   AN_1000A_SPL : REAL := 35.0;
   AN_1000A_STOP_TMR : TIMER := (PRE := 10000);
   AN_1000B : CM_AI_SCL := (RawMin := 4000, RawMax := 20000, EuMax := 1000.0, In_Raw := 5314, Percent := 8.2125, PV := 82.125);
   AN_1000B_RESTART_TMR : TIMER := (PRE := 10000);
   AN_1000B_SP : REAL := 200.0;
   AN_1000B_SPL : REAL := 140.0;
   AN_1000B_STOP_TMR : TIMER := (PRE := 10000);
   AN_1000C : CM_AI_SCL := (RawMin := 4000, RawMax := 20000, EuMin := -85.0, EuMax := 70.0, In_Raw := 4832, Percent := -109.91429, PV := -76.94);
   AN_1000C_RESTART_TMR : TIMER := (PRE := 10000);
   AN_1000C_SP : INT := -69;
   AN_1000C_STOP_TMR : TIMER := (PRE := 10000);
   AN_101_PERMISSIVE_AUTO : BOOL;   // Does the PLC look at AN-101
   AN_101A : CM_AI_SCL := (RawMin := 4000, RawMax := 20000, EuMax := 1000.0, In_Raw := 4241, Percent := 1.50625, PV := 15.0625);
   AN_101A_RESTART_TIME : REAL := 30.0;
   AN_101A_RESTART_TMR : TIMER := (PRE := 30000);
   AN_101A_SP : REAL := 40.0;
   AN_101A_STOP_TIME : REAL := 10.0;
   AN_101A_STOP_TMR : TIMER := (PRE := 10000);
   AN_101B : CM_AI_SCL := (RawMin := 4000, RawMax := 20000, EuMax := 1000.0, In_Raw := 3716, Percent := -1.7750001, PV := -17.75);
   AN_101B_RESTART_TIME : REAL := 30.0;
   AN_101B_RESTART_TMR : TIMER := (PRE := 30000);
   AN_101B_SP : REAL := 40.0;
   AN_101B_STOP_TIME : REAL := 10.0;
   AN_101B_STOP_TMR : TIMER := (PRE := 10000);
   AN_101C : CM_AI_SCL := (RawMin := 4000, RawMax := 20000, EuMax := 1000.0, In_Raw := 4014, Percent := 0.087500006, PV := 0.875);
   AN_101C_RESTART_TIME : REAL := 10.0;
   AN_101C_RESTART_TMR : TIMER := (PRE := 10000);
   AN_101C_SP : REAL := 1001.0;
   AN_101C_STOP_TIME : REAL := 1000.0;
   AN_101C_STOP_TMR : TIMER := (PRE := 1000000);
   AN_200A : CM_AI_SCL := (RawMax := 10000, EuMax := 5000.0, In_Raw := 4, Percent := 0.04, PV := 2.0);
   AN_200A_RESTART_TMR : TIMER := (PRE := 10000);
   AN_200A_SP : REAL := 30.0;
   AN_200A_STOP_TMR : TIMER := (PRE := 2000);
   ARGON_FROM_TK1100A : BOOL := 1;
   ARGON_FROM_TK700 : BOOL;
   ARS14002_PLC_LEDStatus : INT := 3;
   ARS14002_PLC_Slot1Status : INT := 16384;
   ARS14002_PLC_Slot2Status : INT := 16384;
   ARS14002_PLC_Slot3Status : INT := 16384;
   ARS14002_PLC_Slot4Status : INT := 16384;
   ARS14002_PLC_Slot5Status : INT := 16384;
   ARS14002_PLC_Status : INT := 12384;
   ARS_AUTORETURN_IGNORE_AUTO : BOOL;   // Turns furnace return autoswitch on or off
   ARS_COLLECT : BOOL;
   ARS_COLLECT_AUTO : BOOL;
   ARS_DERIME_AUTO : BOOL := 1;
   ARS_DERIME_AUTO_OSF_OB : BOOL;
   ARS_DERIME_AUTO_OSF_SB : BOOL := 1;
   ARS_FULL_COLLECTION : BOOL;
   ARS_FULL_COLLECTION_LATCH : BOOL;   // LATCHES THE FIRST TIME ARS HITS FULL COLLECTION DURING A MODE_ATOMIZE
   ARS_FULL_COLLECTION_TMR : TIMER := (PRE := 10000);
   ARS_IDLE : BOOL := 1;   // **future use
   ARS_Manual_Backfill : BOOL;   // **future use
   ARS_READY_TO_RECEIVE : BOOL;
   ARS_READY_TO_SEND : BOOL;
   ARS_READY_TO_SEND_TMR : TIMER := (PRE := 5000, ACC := 5000, EN := 1, DN := 1);
   ARS_RETURN : BOOL;
   ARS_RETURN_AUTO : BOOL := 1;
   ARS_SOURCE_SWITCH_AUTO : BOOL;   // Switch between TK-700 and TK-1100A
   ARS_STANDBY : BOOL;
   ARS_StartRecycle : TIMER := (PRE := 2000);
   ARS_TO_AT3 : UDT_IPC := (ConnectionStatus.RunMode := 1, REAL[0] := 1.2493749, REAL[1] := 0.63687515, REAL[2] := 1.2575002, REAL[4] := 2394.8313, REAL[5] := 2228.625, REAL[6] := -1.03125, REAL[7] := 53.200012, REAL[8] := 82.125, REAL[9] := 12.3, REAL[10] := 2.0, REAL[11] := 15.0625, REAL[12] := -17.8125, REAL[13] := 0.875, REAL[14] := -1.63125, REAL[15] := -0.19375, REAL[16] := 0.6625, REAL[17] := -0.03125, REAL[18] := 5.275, REAL[19] := 1.25, REAL[20] := 248.67676); {produced}
   AT2_ATOMIZE_FLOW : REAL := 0.009765923;
   AT2_ATOMIZE_FLOW_ATOMIZE_SP : REAL := 30.0;
   AT2_ATOMIZE_FLOW_SCFM : REAL := 0.094368115;
   AT2_ATOMIZE_LATCH : BOOL;
   AT2_ATOMIZE_VALVE_OPEN : BOOL;
   AT2_AtomizingStatus_OSF_OB : BOOL;
   AT2_AtomizingStatus_OSF_SB : BOOL;
   AT2_AtomizingStatus_OSR_OB : BOOL;
   AT2_AtomizingStatus_OSR_SB : BOOL;
   AT2_CHAMBER_PRESSURE : REAL := -0.6632662;
   AT2_CHAMBER_PRESSURE_SP : REAL := -10.5;
   AT2_COMM_STATUS_CONS : BOOL := 1;
   AT2_COMM_STATUS_PROD : BOOL := 1;
   AT2_END_ATOMIZATION : BOOL;
   AT2_FT_202_TOTAL_HEAT : REAL := 26243.87;
   AT2_HIBON_DISCHARGE_TEMP : REAL := 76.04429;
   AT2_HIBON_DISCHARGE_TEMP_MAX : REAL := 262.64694;
   AT2_HIBON_INSERTION_VALVE_OPEN : BOOL;
   AT2_HIBON_RUNNING : BOOL;
   AT2_INLET_FLOW : REAL := -0.59600025;
   AT2_INLET_FLOW_BACKFILL_SP : REAL := 15.0;
   AT2_INLET_FLOW_SCFM : REAL := -5.7591505;
   AT2_INLET_VALVE_OPEN : BOOL;
   AT2_MELT_STATUS : BOOL;
   AT2_NONATOMIZE_FLOW : REAL := -7.5225983;
   AT2_PARTICULATE_POST_CYCLONE : REAL := 1.0125608;
   AT2_PARTICULATE_POST_FILTER : REAL;
   AT2_PEDESTAL_LEVEL : REAL := 0.9041128;
   AT2_PLANT_ATOMIZING : BOOL;
   AT2_PLANT_ATOMIZING_ONS : BOOL;
   AT2_PLANT_BACKFILL : BOOL;
   AT2_PLANT_BACKFILL_TIMEOUT_TMR : TIMER := (PRE := 1800000);
   AT2_PLANT_COLLECT_AUTO : BOOL;
   AT2_PLANT_COLLECTING : BOOL;
   AT2_PLANT_COLLECTION_PERCENT : REAL := 88.49419;
   AT2_PLANT_COLLECTION_PERCENT_GOOD_GAS : REAL := 90.52875;
   AT2_PLANT_COLLECTION_TIME : TIMER := (PRE := 6000000, ACC := 1011437);
   AT2_PLANT_COMMLOSS : BOOL;
   AT2_PLANT_END_ATOMIZATION_TMR : TIMER := (PRE := 5000);   // WAIT AFTER ATOMIZATION END SIGNAL
   AT2_PLANT_GOOD_GAS_PERCENT : REAL := 96.67721;
   AT2_PLANT_GOOD_GAS_TIME : TIMER := (PRE := 7200000, ACC := 1117255);   // AT2 total time with good gas and no collection stops
   AT2_PLANT_GOOD_H2O_PERCENT : REAL := 99.13469;
   AT2_PLANT_GOOD_H2O_TIME : TIMER := (PRE := 7200000, ACC := 1145655);   // AT2 time with good dew point and no collection stop
   AT2_PLANT_GOOD_O2_PERCENT : REAL := 96.67721;
   AT2_PLANT_GOOD_O2_TIME : TIMER := (PRE := 7200000, ACC := 1117255);   // AT2 time with good O2 and no collection stop
   AT2_PLANT_H2O_MIN : REAL := -81.8225;   // AT2 Heat Minimum after burp
   AT2_PLANT_LIKELY_COLLECTING : BOOL;
   AT2_PLANT_LIKELY_COLLECTION_TIME : TIMER := (PRE := 6000000, ACC := 1033938);
   AT2_PLANT_MAX_H2O : REAL := -81.541565;
   AT2_PLANT_MAX_O2 : REAL := 41.0;
   AT2_PLANT_O2_MIN : REAL := 15.5;   // AT2 Heat Minimum after burp
   AT2_PLANT_POST_ATOMIZE_TON : TIMER := (PRE := 1800000, ACC := 1800000, EN := 1, DN := 1);
   AT2_PLANT_POST_ATOMIZING : BOOL := 1;
   AT2_PLANT_POST_ATOMIZING_CHAMBER_SP : REAL := -3.0;
   AT2_PLANT_POST_ATOMIZING_TON : BOOL;
   AT2_PLANT_POST_HEAT_NOTIFICATION_TON : TIMER := (PRE := 10000, ACC := 10000, EN := 1, DN := 1);
   AT2_PLANT_RETURN_AUTO : BOOL := 1;
   AT2_PRAXAIR_PRESSURE : REAL := -1101.6534;
   AT2_PRAXAIR_PRESSURE_RETURN_SPH : REAL := 4200.0;
   AT2_PRAXAIR_PRESSURE_RETURN_SPL : REAL := 3400.0;
   AT2_PRESTART : BOOL;
   AT2_PT_101B_Pressure_Override : REAL := 4.0;   // Setpoint at which FCV_101 will open and relieve the pressure despite controls, not an interlock
   AT2_START_ATOMIZATION : BOOL;
   AT2_V1_NOT_OPEN_ONS : BOOL;
   AT2_V1_OPEN : BOOL;
   AT2_V1_OPEN_OSR_OB : BOOL;
   AT2_V1_OPEN_OSR_SB : BOOL;
   AT2_V1_OPEN_POSTHEAT_CTR : COUNTER := (PRE := 100, ACC := 14);
   AT2_V1_OPEN_POSTHEAT_CTR_SP : DINT := 5;
   AT2_V4_OPEN : BOOL;
   AT3_ATOMIZE_FLOW : REAL := 0.046901885;
   AT3_ATOMIZE_FLOW_ATOMIZE_SP : REAL := 30.0;
   AT3_ATOMIZE_FLOW_SCFM : REAL := 0.5414932;
   AT3_ATOMIZE_VALVE_OPEN : BOOL;
   AT3_AtomizingStatus_OSF_OB : BOOL;
   AT3_AtomizingStatus_OSF_SB : BOOL;
   AT3_AtomizingStatus_OSR_OB : BOOL;
   AT3_AtomizingStatus_OSR_SB : BOOL;
   AT3_CHAMBER_PRESSURE : REAL := 0.15592758;
   AT3_CHAMBER_PRESSURE_SP : REAL := -10.5;
   AT3_CHAMBER_VACUUM : REAL := -1.0;
   AT3_COMM_STATUS_CONS : BOOL := 1;
   AT3_COMM_STATUS_PROD : BOOL := 1;
   AT3_END_ATOMIZATION : BOOL;
   AT3_FT_202_TOTAL_HEAT : REAL;
   AT3_HIBON_DISCHARGE_TEMP : REAL := 68.16922;
   AT3_HIBON_DISCHARGE_TEMP_MAX : REAL := 268.5566;
   AT3_HIBON_INSERTION_VALVE_OPEN : BOOL;
   AT3_HIBON_RUNNING : BOOL;
   AT3_INLET_FLOW : REAL := 0.05965271;
   AT3_INLET_FLOW_BACKFILL_SP : REAL := 15.0;
   AT3_INLET_FLOW_SCFM : REAL := 0.5975359;
   AT3_INLET_VALVE_OPEN : BOOL;
   AT3_MELT_STATUS : BOOL;
   AT3_NONATOMIZE_FLOW : REAL := 1.0296371;
   AT3_PARTICULATE_POST_CYCLONE : REAL := 0.12207031;
   AT3_PARTICULATE_POST_FILTER : REAL;
   AT3_PEDESTAL_LEVEL : REAL;
   AT3_PLANT_ATOMIZING : BOOL;
   AT3_PLANT_ATOMIZING_ONS : BOOL;
   AT3_PLANT_BACKFILL : BOOL;
   AT3_PLANT_BACKFILL_TIMEOUT_TMR : TIMER := (PRE := 1800000);
   AT3_PLANT_COLLECT_AUTO : BOOL;
   AT3_PLANT_COLLECTING : BOOL;
   AT3_PLANT_COLLECTION_PERCENT : REAL := 48.725945;
   AT3_PLANT_COLLECTION_PERCENT_GOOD_GAS : REAL := 71.160706;
   AT3_PLANT_COLLECTION_TIME : TIMER := (PRE := 6000000, ACC := 567592);
   AT3_PLANT_COMMLOSS : BOOL;
   AT3_PLANT_GOOD_GAS_PERCENT : REAL := 63.344948;
   AT3_PLANT_GOOD_GAS_TIME : TIMER := (PRE := 7200000, ACC := 797620);   // total time with good gas and no collection stops
   AT3_PLANT_GOOD_H2O_PERCENT : REAL := 99.205826;
   AT3_PLANT_GOOD_H2O_TIME : TIMER := (PRE := 7200000, ACC := 1249169);   // time with good dew point and no collection stop
   AT3_PLANT_GOOD_O2_PERCENT : REAL := 63.344948;
   AT3_PLANT_GOOD_O2_TIME : TIMER := (PRE := 7200000, ACC := 797620);   // time with good O2 and no collection stop
   AT3_PLANT_H2O_MIN : REAL := -83.692184;   // AT3 Plant Minimum after burp
   AT3_PLANT_LIKELY_COLLECTING : BOOL;
   AT3_PLANT_LIKELY_COLLECTION_TIME : TIMER := (PRE := 6000000, ACC := 659492);
   AT3_PLANT_MAX_H2O : REAL := -82.34563;
   AT3_PLANT_MAX_O2 : REAL := 41.5;
   AT3_PLANT_O2_MIN : REAL := 8.0;   // AT3 Plant Minimum after burp
   AT3_PLANT_POST_ATOMIZE_TON : TIMER := (PRE := 1800000, ACC := 1800000, EN := 1, DN := 1);
   AT3_PLANT_POST_ATOMIZING : BOOL := 1;
   AT3_PLANT_POST_ATOMIZING_CHAMBER_SP : REAL := -3.0;
   AT3_PLANT_POST_HEAT_NOTIFICATION_TON : TIMER := (PRE := 10000, ACC := 10000, EN := 1, DN := 1);
   AT3_PLANT_RETURN_AUTO : BOOL := 1;
   AT3_PRESTART : BOOL;
   AT3_PT_101C_Press_Override : REAL := 4.0;   // Pressure at which FCV101 will open despite the control scheme, not an interlock
   AT3_START_ATOMIZATION : BOOL;
   AT3_TO_ARS : UDT_IPC := (ConnectionStatus.RunMode := 1, BOOL[0] := 1, BOOL[10] := 1, BOOL[11] := 1, REAL[10] := -0.59600025, REAL[11] := 0.009765923, REAL[12] := 76.04429, REAL[13] := 0.9041128, REAL[14] := -0.6632662, REAL[15] := -1114.4707, REAL[17] := 1.0125608, REAL[20] := 0.061017055, REAL[21] := 0.054569516, REAL[22] := 68.1691, REAL[23] := -0.00041597337, REAL[24] := 0.15122452, REAL[25] := -1.0, REAL[27] := 0.12207031);
   AT3_V1_OPEN : BOOL;
   AT3_V1_OPEN_OSR_OB : BOOL;
   AT3_V1_OPEN_OSR_SB : BOOL;
   AT3_V1_OPEN_POSTHEAT_CTR : COUNTER := (PRE := 100, ACC := 14);
   AT3_V4_OPEN : BOOL;
   Auto_CP_Select_HMI : BOOL;
   Auto_CP_Select_Inactive_ONS : BOOL := 1;
   BACKFILL_PAUSE_BLOWBACK_ONS : BOOL;
   BLENDING_OVERRIDE : BOOL := 1;
   BLOWBACK_COMMAND : BOOL;
   BLOWBACK_COUNTER : COUNTER := (PRE := 3);
   BLOWBACK_PRESS_SPH : REAL := 8.0;
   BLOWBACK_PRESS_SPL : REAL := 1.3;
   BLOWBACK_PRESS_UNSAFE : REAL := 9.5;
   BLOWBACK_REQUEST : BOOL;
   BLOWBACK_REQUEST_OFF_ONS : BOOL := 1;
   BLOWBACK_REQUEST_ONS : BOOL;
   BLOWBACKS_REQUESTED : DINT := 3;
   BNOT_1002 : FBD_BOOLEAN_NOT := (Out := 1);
   CALC_AN_1000B_BLENDED : REAL := 82.125;
   Calc_Day : INT;
   CALC_FT_1002_MONTH_RETURN : REAL;
   CALC_FT_1002_MONTH_TOTALIZER : TOTALIZER := (In := -1.03125, TimeBase := 1, Gain := 1.0, ProgProgReq := 1, ProgStopReq := 1, RTSTime := 1, OldTotal := 15819730.0, ProgOper := 1, TargetFlag := 1, TargetDev1Flag := 1, TargetDev2Flag := 1, LowInCutoffFlag := 1, DeltaT := 0.001);
   CALC_FT_1002_MONTH_TOTALIZER1 : TOTALIZER := (Gain := 1.0, RTSTime := 1);
   CALC_FT_1002_MONTH_TOTALIZER_RESET : BOOL;
   CALC_FT_1002_MONTH_TOTALIZER_START : BOOL;
   CALC_FT_1002_MONTH_TOTALIZER_STOP : BOOL := 1;
   Calc_FT_1002_Return_Total : DINT[2100,13] := ([2018,5] := 134676, [2018,6] := 409656, [2018,7] := 822706, [2018,8] := 599070, [2018,9] := 3547396, [2018,10] := 3647326, [2018,11] := 3203450, [2018,12] := 3276487, [2019,1] := 6793074, [2019,2] := 10828261, [2019,3] := 18080340, [2019,4] := 11366855, [2019,5] := 9161697, [2019,6] := 12851823, [2019,7] := 12738279, [2019,8] := 15393065, [2019,9] := 13514600, [2019,10] := 15668862, [2019,11] := 10873787, [2019,12] := 10924969, [2020,1] := 13740664, [2020,2] := 17859208, [2020,3] := 17781294, [2020,4] := 15819730);
   CALC_FT_1002_TOTAL_RETURN : REAL := 14241.822;
   CALC_FT_1002_TOTALIZER_RETURN : TOTALIZER := (In := -1.03125, TimeBase := 1, Gain := 1.0, ProgProgReq := 1, ProgStopReq := 1, RTSTime := 1, Total := 14241.822, OldTotal := 26887.246, ProgOper := 1, TargetFlag := 1, TargetDev1Flag := 1, TargetDev2Flag := 1, LowInCutoffFlag := 1, DeltaT := 0.001);
   CALC_FT_202_MONTH : REAL := 7071.2705;
   CALC_FT_202_MONTH_TOTALIZER : TOTALIZER := (TimeBase := 1, Gain := 1.0, ProgProgReq := 1, ProgStartReq := 1, RTSTime := 1, Total := 7071.2705, OldTotal := 12203607.0, ProgOper := 1, RunStop := 1, TargetFlag := 1, TargetDev1Flag := 1, TargetDev2Flag := 1, LowInCutoffFlag := 1, DeltaT := 0.001);
   CALC_FT_202_TOTAL_HEAT : REAL := 26243.87;
   CALC_FT_202_TOTALIZER : TOTALIZER := (TimeBase := 1, Gain := 1.0, ProgProgReq := 1, ProgStopReq := 1, RTSTime := 1, Total := 26243.87, OldTotal := 26411.75, ProgOper := 1, TargetFlag := 1, TargetDev1Flag := 1, TargetDev2Flag := 1, LowInCutoffFlag := 1, DeltaT := 0.001);
   CALC_FT_202_TOTALIZER1 : TOTALIZER := (Gain := 1.0, RTSTime := 1);
   CALC_FT_202_TOTALIZER_AT2 : TOTALIZER := (TimeBase := 1, Gain := 1.0, ProgProgReq := 1, ProgStopReq := 1, RTSTime := 1, Total := 26243.87, ProgOper := 1, TargetFlag := 1, TargetDev1Flag := 1, TargetDev2Flag := 1, LowInCutoffFlag := 1, DeltaT := 0.001);
   CALC_FT_202_TOTALIZER_AT3 : TOTALIZER := (TimeBase := 1, Gain := 1.0, ProgProgReq := 1, ProgStopReq := 1, RTSTime := 1, OldTotal := 26411.75, ProgOper := 1, TargetFlag := 1, TargetDev1Flag := 1, TargetDev2Flag := 1, LowInCutoffFlag := 1, DeltaT := 0.001);
   CALC_FT_202_TOTALIZER_PILOT : TOTALIZER := (TimeBase := 1, Gain := 1.0, ProgProgReq := 1, ProgStopReq := 1, RTSTime := 1, ProgOper := 1, TargetFlag := 1, TargetDev1Flag := 1, TargetDev2Flag := 1, LowInCutoffFlag := 1, DeltaT := 0.001);
   CALC_HMI_FLOW : REAL;
   Calc_Month : INT := 5;
   CALC_NEXT_DAY_OSR_OB : BOOL;
   CALC_NEXT_DAY_OSR_SB : BOOL;
   CALC_NEXT_MONTH_OSR_OB : BOOL;
   CALC_NEXT_MONTH_OSR_SB : BOOL := 1;
   Calc_TK_700_Fill_Lvl : REAL;
   Calc_TK_700_Fill_Start_Lvl : REAL;
   Calc_TK_700_Fill_Stop_Lvl : REAL;
   Calc_TK_700_Fill_Total : DINT[2100,13] := ([2018,6] := 49577, [2018,7] := 6585, [2018,8] := 28493, [2018,9] := 140310, [2018,10] := 25327, [2018,11] := 3926, [2019,3] := 570, [2019,4] := 3166, [2019,5] := 190, [2019,8] := 39320, [2020,1] := 4749);
   Calc_TK_700_Month_Fill : REAL;
   Calc_TK_700_Month_Totalizer_Reset : BOOL;
   Calc_TK_700_Month_Totalizer_Start : BOOL;
   Calc_TK_700_Month_Totalizer_Stop : BOOL := 1;
   Calc_Year : INT := 2020;
   Cold_Box_Idle : BOOL := 1;   // **future use
   COLDBOX_IDLE : BOOL;
   COLDBOX_REACTION_TMR : TIMER := (PRE := 3600000, ACC := 78224);
   COLDBOX_REACTION_TMR_SEC : REAL := 78.22401;
   COLDBOX_STANDBY : BOOL;
   Collect_Stop_AT2_O2 : BOOL;
   Collect_Stop_AT3_O2 : BOOL;
   Collect_Stop_Dew_Pt : BOOL;
   COLLECT_STOP_INIT : TIMER := (PRE := 2000, ACC := 2000, EN := 1, DN := 1);
   Collect_Stop_O2 : BOOL;
   Collect_Stop_PILOT_O2 : BOOL;
   COLLECTION_ESTIMATE_SCALING_FACTOR : REAL;
   COLLECTION_LIKELY_PERCENTAGE : REAL := 0.5;
   Cooldown_Complete_ONS_OB : BOOL;
   Cooldown_Complete_ONS_SB : BOOL;
   COOLDOWN_CYCLES_MIN : DINT[10] := ([0] := 16, [1] := 16, [2] := 16, [3] := 8, [4] := 4, [5] := 1, [6] := 20, [7] := 8, [8] := 5, [9] := 10);
   COOLDOWN_CYCLES_SEC : DINT[10] := ([0] := 47, [1] := 47, [2] := 47, [3] := 3, [4] := 5, [5] := 52, [6] := 19, [7] := 52, [8] := 10, [9] := 59);
   COOLDOWN_TIMER1 : TIMER := (PRE := 99999999, ACC := 1007975);
   COOLDOWN_TIMER1_MIN : DINT := 16;
   COOLDOWN_TIMER1_MS : DINT := 47975;
   COOLDOWN_TIMER1_SEC : DINT := 47;
   CP_Auto : BOOL := 1;
   CP_Auto_ONS : BOOL;
   CP_Hi_Press_Shutoff : BOOL;
   CP_PID_MaxOut : REAL := 60.0;
   CP_PumpUp : BOOL;
   CP_PumpUp_DN_ONS_OB : BOOL;
   CP_PumpUp_PressurePermissive : BOOL := 1;
   CP_PumpUp_Standby_Press_SP_H : DINT := 5000;
   CP_PumpUp_Standby_Press_SP_L : DINT := 4500;
   CP_Run : BOOL;
   CP_Run_Atomize : BOOL;
   CP_Run_ONS_OB : BOOL;
   CP_Run_ONS_SB : BOOL;
   CP_Run_Standby : BOOL;
   CP_RUN_TIMESTAMP_DAY : DINT[10] := ([0] := 26, [1] := 26, [2] := 26, [3] := 26, [4] := 26, [5] := 26, [6] := 26, [7] := 26, [8] := 26, [9] := 26);
   CP_RUN_TIMESTAMP_HOUR : DINT[10] := ([0] := 10, [1] := 10, [2] := 10, [3] := 10, [4] := 6, [5] := 5, [6] := 3, [7] := 3, [8] := 3);
   CP_RUN_TIMESTAMP_MIN : DINT[10] := ([0] := 33, [1] := 33, [2] := 33, [3] := 33, [4] := 36, [5] := 36, [6] := 22, [7] := 22, [8] := 22, [9] := 29);
   CP_RUN_TIMESTAMP_MONTH : DINT[10] := ([0] := 4, [1] := 4, [2] := 4, [3] := 4, [4] := 4, [5] := 4, [6] := 4, [7] := 4, [8] := 4, [9] := 4);
   CP_RUN_TIMESTAMP_SEC : DINT[10] := ([0] := 50, [1] := 50, [2] := 50, [3] := 50, [4] := 27, [5] := 11, [6] := 20, [7] := 20, [8] := 20, [9] := 22);
   CP_RUN_TIMESTAMP_YEAR : DINT[10] := ([0] := 2020, [1] := 2020, [2] := 2020, [3] := 2020, [4] := 2020, [5] := 2020, [6] := 2020, [7] := 2020, [8] := 2020, [9] := 2020);
   CP_Select_Auto : BOOL;
   CP_Select_Auto_ONS : BOOL;
   CP_Speed_SP_Atomize : REAL := 20.0;
   CP_Speed_SP_Standby : DINT := 60;
   CP_Speed_Start_Recycle : REAL := 15.0;
   CP_Start_Vent_TMR_PRE : DINT := 45000;
   CP_Stop : BOOL := 1;
   CP_Stop_ONS_OB : BOOL;
   CP_Stop_ONS_SB : BOOL := 1;
   CP_System_Down : BOOL;   // Catch all bit for pump problems for ARS ready to send
   CYCLE_TIME_AT2_MIN : DINT := 180;
   CYCLE_TIME_AT3_MIN : DINT := 180;
   CYCLE_TIME_PILOT_MIN : DINT := 180;
   CYCLE_TIME_REM_AT2_MIN : REAL;
   CYCLE_TIME_REM_AT3_MIN : REAL;
   CYCLE_TIME_REM_PILOT_MIN : REAL;
   DC_OK_1000 : BOOL := 1;
   DC_OK_600 : BOOL := 1;
   DC_OK_800 : BOOL := 1;
   DC_OK_MCP : BOOL := 1;
   DEL_FCV_1002_FLOW_SP_AUTO : REAL;
   DELETE_REAL_BLOWBACKS_REQUESTED : REAL := 3.0;
   DEOXO_ARGON_PURGE_DEPRESS : BOOL;
   DEOXO_ARGON_PURGE_FILL : BOOL;
   DEOXO_ARGON_PURGE_HIFLOW : BOOL;
   DEOXO_ARGON_PURGE_LOFLOW : BOOL;
   Deoxo_CurrentState : DINT;
   DEOXO_DEPRESS_TON : TIMER := (PRE := 500);
   DEOXO_DRY_REM : DINT;
   DEOXO_DRY_TON : TIMER := (PRE := 1800000);
   DEOXO_EXOTHERM_SP : REAL := 250.0;
   DEOXO_OVERTEMP : BOOL;
   DEOXO_OVERTEMP_SPH : REAL := 375.0;
   DEOXO_OVERTEMP_SPL : REAL := 300.0;
   DEOXO_POST_EXO_REM : DINT;
   DEOXO_POST_EXOTHERM_TON : TIMER := (PRE := 1800000);
   DEOXO_PREHEAT_SP : REAL := 150.0;
   DEOXO_PURGE_CYC_REM : DINT := 7;
   DEOXO_PURGE_CYCLE_CTU : COUNTER := (PRE := 7);
   DEOXO_REGEN_HMI_BIT : BOOL;
   DEOXO_REGEN_HMI_BIT_ONS_F : BOOL := 1;
   DEOXO_REGEN_HMI_BIT_ONS_R : BOOL;
   DEOXO_REGEN_RESET : BOOL;
   DEOXO_REGEN_RESET_ONS : BOOL;
   DEOXO_REGEN_RUN : BOOL;
   DEOXO_REGEN_START_PB : BOOL;
   DEOXO_REGEN_STOP_PB : BOOL;
   Deoxo_TransitionState : DINT;
   DEOXO_VENT_SPL : REAL := 3.0;
   DEOXO_VENT_SWITCH_SP : REAL := 100.0;
   DERIME_HOLD : BOOL;
   DERIME_HP_CYCLE : BOOL := 1;
   DERIME_HP_SPH : REAL := 30.0;   // SETPOINT FOR VALVES BESIDES FCV-202
   DERIME_HP_SPL : REAL := 1.3;   // SETPOIT FOR VALVES BESIDES FCV-202
   EN_1250 : BOOL;   // HXR-1250 Enable Signal
   ESTOP_1 : BOOL := 1;   // Pump Skid E-Stops
   ESTOP_2 : BOOL := 1;   // FAN/HXR E-Stops
   ESTOP_HMI : BOOL;
   ESTOP_PL : CM_DO_GENERIC := (Auto := 1);
   ESTOP_ResetReq : BOOL;
   ESTOP_TRIP : BOOL;
   ew_test2 : BOOL;
   EW_TEST_101 : BOOL;
   ew_test_102 : BOOL := 1;
   ew_test_200 : BOOL;
   EW_TEST_ATOMIZE : BOOL;
   EW_TEST_FIRSTSCAN : BOOL;
   EW_TEST_FVR800C : BOOL;
   EW_TEST_FVR800D : BOOL;
   ew_TEST_P800A_LOCKOUT : BOOL;
   EW_TEST_VFD800A : BOOL;
   EW_TEST_VFD800B : BOOL;
   EW_TEST_VFDSPD : BOOL;
   FCV_1001 : CM_AO_VLV := (EuMax := 100.0, RawMin := 4000, RawMax := 20000, ZT := 98.85, EngValue := 100.0, Out_Raw := 20000, Alm_Dev_SP := 10.0, Alm_Dev_TmrPre := 10);
   FCV_1001_ENABLE_TON : TIMER := (PRE := 2000, ACC := 2000, EN := 1, DN := 1);
   FCV_1001_STARTPOS : REAL := 20.0;
   FCV_1002 : CM_AO_VLV := (EuMax := 100.0, RawMin := 4000, RawMax := 20000, ZT := 35.21875, EngValue := 30.0, Out_Raw := 8800, Alm_Dev_SP := 10.0, Alm_Dev_TmrPre := 10);
   FCV_1002_Atomize_Mode : BOOL;
   FCV_1002_FLOW_MODE : BOOL;   // 1 = FLOW CONTROL FT-1002 0 = PRESSURE CONTROL PT-1003
   FCV_1002_FLOW_MODE_AN_100B_PPM_MAX : REAL := 300.0;
   FCV_1002_FLOW_MODE_MIN_FLOW : REAL := 800.0;
   FCV_1002_FLOW_MODE_N2_PPM_SP : REAL := 150.0;
   FCV_1002_FLOW_NOT_ATOMIZE_SP : REAL := 400.0;
   FCV_1002_FLOW_SP : REAL := 850.0;
   FCV_1002_FLOW_SP_AUTO : BOOL;
   FCV_1002_HIGHPRESS_MAXOPEN : REAL := 27.0;
   FCV_1002_PT_1003_HIGHALM : BOOL;
   FCV_1002_PT_1003_HIGHLIM : REAL := 2450.0;
   FCV_1002_PT_1003_HIGHLIM_RESET : REAL := 2400.0;
   FCV_1002_PVSWITCH_AUTO : BOOL := 1;
   FCV_1002_SP_Atomize : REAL := 2350.0;
   FCV_1002_SP_Idle_Standby : REAL := 2350.0;
   FCV_1002_STARTPOS : REAL := 40.0;
   FCV_101A : CM_AO_VLV := (FailPos := 1, EuMax := 100.0, RawMin := 4000, RawMax := 20000, ZT := -0.03125, Out_Raw := 20000, Alm_Dev_SP := 10.0, Alm_Dev_TmrPre := 60);
   FCV_101A_COLLECTION_CV_LOW : REAL := 20.0;
   FCV_101A_DLA : REAL := 60.0;
   FCV_101A_DLA_BUMP_TMR : TIMER := (PRE := 2000);
   FCV_101A_DLA_TMR : TIMER := (PRE := 60000);
   FCV_101A_STARTPOS : REAL := 60.0;
   FCV_101A_ZT_OSR : BOOL;
   FCV_101B : CM_AO_VLV := (FailPos := 1, EuMax := 100.0, RawMin := 4000, RawMax := 20000, ZT := 5.275, Out_Raw := 20000, Alm_Dev_SP := 12.0, Alm_Dev_TmrPre := 30);
   FCV_101B_COLLECTION_CV_LOW : REAL := 20.0;
   FCV_101B_DLA : REAL := 45.0;
   FCV_101B_DLA_BUMP_TMR : TIMER := (PRE := 2000);
   FCV_101B_DLA_TMR : TIMER := (PRE := 45000);
   FCV_101B_STARTPOS : REAL := 60.0;
   FCV_101B_ZT_OSR : BOOL;
   FCV_101C : CM_AO_VLV := (FailPos := 1, EuMax := 100.0, RawMin := 4000, RawMax := 20000, ZT := 1.24375, Out_Raw := 20000, Alm_Dev_SP := 10.0, Alm_Dev_TmrPre := 30);
   FCV_101C_COLLECTION_CV_LOW : REAL := 20.0;
   FCV_101C_DLA : REAL := 60.0;
   FCV_101C_DLA_BUMP_TMR : TIMER := (PRE := 2000);
   FCV_101C_DLA_TMR : TIMER := (PRE := 60000);
   FCV_101C_STARTPOS : REAL := 60.0;
   FCV_101C_ZT_OSR : BOOL;
   FCV_102A : CM_AO_VLV := (FailPos := 1, EuMax := 100.0, RawMin := 4000, RawMax := 20000, ZT := -0.01875, Out_Raw := 20000, Alm_Dev_SP := 10.0, Alm_Dev_TmrPre := 5);
   FCV_102A_AT_STARTPOS : BOOL;
   FCV_102A_COLLECTION_CV_HIGH : REAL := 6.0;
   FCV_102A_SP_Atomize_Venting : REAL := 0.8;
   FCV_102A_SP_Idle_Collecting : REAL := 1.5;
   FCV_102A_STARTPOS : REAL := 50.0;
   FCV_102A_STARTPOS_TIMEOUT : TIMER := (PRE := 600000);
   FCV_102B : CM_AO_VLV := (FailPos := 1, EuMax := 100.0, RawMin := 4000, RawMax := 20000, ZT := -1.63125, EngValue := 4.0, Out_Raw := 19360, Alm_Dev_SP := 20.0, Alm_Dev_TmrPre := 60);
   FCV_102B_AT_STARTPOS : BOOL;
   FCV_102B_CLOSE_DLA_PRE : REAL := 180.0;
   FCV_102B_CLOSE_DLA_TMR : TIMER := (PRE := 180000);
   FCV_102B_COLLECTION_CV_HIGH : REAL := 6.0;
   FCV_102B_SP_Atomize_Venting : REAL := 0.5;
   FCV_102B_SP_Idle_Collecting : REAL := 1.5;
   FCV_102B_STARTPOS : REAL := 50.0;
   FCV_102B_STARTPOS_TIMEOUT : TIMER := (PRE := 600000);
   FCV_102C : CM_AO_VLV := (FailPos := 1, EuMax := 100.0, RawMin := 4000, RawMax := 20000, ZT := -0.19375, EngValue := 0.66082937, Out_Raw := 19894, Alm_Dev_SP := 10.0, Alm_Dev_TmrPre := 60);
   FCV_102C_AT_STARTPOS : BOOL;
   FCV_102C_ATOMIZE_INIT : TIMER := (PRE := 2000);
   FCV_102C_BUMP_CLOSE_POS : REAL := 27.0;
   FCV_102C_BUMPED_CLOSED : BOOL;
   FCV_102C_CLOSE_BUMP_TMR : TIMER := (PRE := 2000);
   FCV_102C_CLOSE_DLA_PRE : REAL;
   FCV_102C_CLOSE_DLA_TMR : TIMER;
   FCV_102C_COLLECTION_CV_HIGH : REAL := 6.0;
   FCV_102C_SP_Atomize_Venting : REAL := 0.5;
   FCV_102C_SP_Idle_Collecting : REAL := 1.5;
   FCV_102C_STARTPOS : REAL := 50.0;
   FCV_102C_STARTPOS_TIMEOUT : TIMER := (PRE := 600000);
   FCV_1221 : CM_AO_VLV := (EuMax := 100.0, RawMin := 4000, RawMax := 20000, ZT := -1.29375, Out_Raw := 4000, Alm_Dev_SP := 10.0, Alm_Dev_TmrPre := 5);
   FCV_1251 : CM_AO_VLV := (EuMax := 100.0, RawMin := 4000, RawMax := 20000, ZT := 2.0875, Out_Raw := 4000, Alm_Dev_SP := 10.0, Alm_Dev_TmrPre := 5);
   FCV_202 : CM_AO_VLV := (EuMax := 100.0, RawMin := 4000, RawMax := 20000, ZT := -0.05625, Out_Raw := 4000, Alm_Dev_SP := 10.0, Alm_Dev_TmrPre := 60);
   FCV_202_BLOWBACK_POS : REAL := 40.0;
   FCV_202_COLLECTION_CERTAIN_SP : REAL := 20.0;
   FCV_202_COLLECTION_CV_LOW : REAL := 20.0;
   FCV_202_COLLECTION_LIKELY_SP : REAL := 20.0;
   FCV_202_HEAT_AVG : REAL := 96.450356;
   FCV_202_HEAT_AVG_TON : TIMER := (PRE := 1000);
   FCV_202_HEAT_TOTAL : REAL := 95871.66;
   FCV_202_OPEN_DLA_PILOT_ADJ : DINT;
   FCV_202_OPEN_DLA_SEC : REAL := 10.0;
   FCV_202_OPEN_DLA_TMR : TIMER := (PRE := 10000);
   FCV_202_OPEN_INIT : TIMER := (PRE := 2000);
   FCV_202_POST_HEAT_VENT_AUTO : BOOL;
   FCV_202_POST_HEAT_VENTS : DINT := 3;
   FCV_202_POST_HEAT_VENTS_CTU : COUNTER;
   FCV_202_PVSWITCH : BOOL;   // 0 = PIT-201 1 = PIT-101C
   FCV_202_SAMPLES : COUNTER := (ACC := 994, DN := 1);
   FCV_202_STARTPOS : REAL := 50.0;
   FCV_204 : CM_AO_VLV := (FailPos := 1, EuMax := 100.0, RawMin := 4000, RawMax := 20000, ZT := 0.55, Out_Raw := 20000, Alm_Dev_SP := 10.0, Alm_Dev_TmrPre := 60);
   FCV_204_AT_STARTPOS : BOOL;
   FCV_204_ATOMIZE_INIT : TIMER := (PRE := 2000);
   FCV_204_COLLECTION_CV_HIGH : REAL := 6.0;
   FCV_204_HEAT_AVG : REAL := 0.07084981;
   FCV_204_HEAT_TOTAL : REAL := 70.42471;
   FCV_204_PVSWITCH : BOOL;   // 0 = PIT-201 1 = PIT-101C
   FCV_204_SP_Atomize : REAL := 1.1;
   FCV_204_SP_Atomize_Venting_Only : REAL := 0.6;
   FCV_204_SP_Idle : REAL := 1.6;
   FCV_204_STARTPOS : REAL := 40.0;
   FCV_204_STARTPOS_0 : REAL;
   FCV_207 : CM_AO_VLV := (EuMax := 100.0, RawMin := 4000, RawMax := 20000, ZT := 0.5125, Out_Raw := 4000, Alm_Dev_SP := 10.0, Alm_Dev_TmrPre := 5);
   FCV_207_BLOWOFF : BOOL;
   FCV_207_FRONT_END_RESCUE : BOOL;
   FCV_207_FRONT_END_RESCUE_AUTO : BOOL := 1;
   FCV_207_FRONT_END_RESCUE_SP : REAL := 0.2;
   FCV_207_POSTHEAT_OFF : BOOL := 1;   // Turn off 207 post heat pressurizing
   FCV_207_POSTHEATPRESSURE : REAL := 0.1;
   FCV_207_POSTHEATPRESSURE_DB : REAL := 0.4;
   FCV_207_PRESSRELIEF_SPH : REAL := 2650.0;
   FCV_207_PRESSRELIEF_SPL : REAL := 2575.0;
   FCV_207_RECYCLEWAITPOS : REAL := 60.0;
   FCV_207_STARTPOS : REAL := 50.0;
   FCV_207_STATICPOS : REAL := 60.0;
   FCV_504 : CM_AO_VLV := (EuMax := 100.0, RawMin := 4000, RawMax := 20000, ZT := 10.00625, EngValue := 10.0, Out_Raw := 5600, Alm_Dev_SP := 10.0, Alm_Dev_TmrPre := 20);
   FCV_504_LOWPRESS_MAXOPEN : REAL := 45.0;
   FCV_504_PT_603_LOLOALM : BOOL;
   FCV_504_PT_603_LOWALM : BOOL;
   FCV_504_PT_603_LOWLIM : REAL := 13.5;
   FCV_504_PT_603_LOWLIM_RESET : REAL := 14.0;
   FCV_504_SP_Atomize : REAL := 23.0;
   FCV_504_SP_Atomize_2Tower : REAL := 15.0;
   FCV_504_SP_Atomize_2Tower_AR : REAL;
   FCV_504_SP_Atomize_2Tower_AR_CALC : REAL;
   FCV_504_SP_Atomize_2Tower_CALC : REAL := 15.0;
   FCV_504_SP_Atomize_AR : REAL := 0.7;
   FCV_504_SP_Atomize_AR_CALC : REAL := 0.7;   // Setpoint with an adjustment for the Pilot Plant
   FCV_504_SP_Atomize_AR_PILOT_ADJ : REAL := -0.2;   // Adjustment for the atomize setpoint on top of what it would be for normal furnaces
   FCV_504_SP_Atomize_CALC : REAL := 23.0;
   FCV_504_SP_Atomize_FRONT_END : REAL := 0.8;
   FCV_504_SP_Atomize_PILOT_ADJ : REAL := -2.6;
   FCV_504_SP_Idle : REAL := 50.0;
   FCV_504_SP_Idle_AR : REAL := 1.5;
   FCV_504_SP_Idle_AR_STORAGE : REAL := 1.5;
   FCV_504_SP_Idle_STORAGE : REAL := 28.0;
   FCV_504_SP_Standby : REAL := 23.0;
   FCV_504_SP_Standby_AR : REAL := 0.3;
   FCV_504_SP_Standby_FRONT_END : REAL := 1.0;
   FCV_504_STARTPOS : REAL := 50.0;
   FCV_603 : CM_AO_VLV := (EuMax := 100.0, RawMin := 4000, RawMax := 20000, ZT := 58.8875, EngValue := 60.0, Out_Raw := 13600, Alm_Dev_SP := 10.0, Alm_Dev_TmrPre := 5);
   FCV_603_Atomize_Start_CV : REAL := 60.0;
   FCV_603_BUMP_TMR : TIMER := (PRE := 2000);
   FCV_603_SP_Atomize : REAL := 120.0;
   FCV_603_SP_Idle : REAL := 120.0;
   FCV_603_SP_Standby : REAL := 120.0;
   FCV_605 : CM_AO_VLV := (EuMax := 100.0, RawMin := 4000, RawMax := 20000, ZT := -0.0375, Out_Raw := 4000, Alm_Dev_SP := 10.0, Alm_Dev_TmrPre := 5);
   FCV_753 : CM_AO_VLV := (EuMax := 100.0, RawMin := 4000, RawMax := 20000, ZT := -0.0125, Out_Raw := 4000, Alm_Dev_SP := 10.0, Alm_Dev_TmrPre := 5);
   FCV_753_SP_Idle : REAL := 4.0;
   FCV_753_SP_Standby : REAL := 4.0;
   FCV_754 : CM_AO_VLV := (EuMax := 100.0, RawMin := 4000, RawMax := 20000, ZT := -1.65625, Out_Raw := 4000, Alm_Dev_SP := 10.0, Alm_Dev_TmrPre := 5);
   FCV_754_SP_Idle : REAL := 24.0;
   FCV_754_SP_Standby : REAL := 22.0;
   FCV_755 : CM_AO_VLV := (EuMax := 100.0, RawMin := 4000, RawMax := 20000, ZT := 3.425, Out_Raw := 4000, Alm_Dev_SP := 10.0, Alm_Dev_TmrPre := 5);
   FCV_STARTPOS_TIMEOUT : TIMER := (PRE := 600000);
   FIRST_SCAN_BIT : BOOL;
   FIT_202_COLLECTION_FLOW : REAL;
   FSL_1000B : BOOL;
   FT_1002 : CM_AI_SCL := (RawMin := 4000, RawMax := 20000, EuMax := 5500.0, In_Raw := 3997, Percent := -0.01875, PV := -1.03125);
   FT_1002_MAVE : REAL := -1.03125;
   FT_1002_MAVE_BLOCK : MOVING_AVERAGE := (In := -1.03125, SampleEnable := 1, NumberOfSamples := 30, Out := -1.03125);
   FT_1002_MAVE_STORAGE : REAL[30] := ([0] := -1.03125, [1] := -1.03125, [2] := -1.03125, [3] := -1.03125, [4] := -1.03125, [5] := -1.03125, [6] := -1.03125, [7] := -1.03125, [8] := -1.03125, [9] := -1.03125, [10] := -1.03125, [11] := -1.03125, [12] := -1.03125, [13] := -1.03125, [14] := -1.03125, [15] := -1.03125, [16] := -1.03125, [17] := -1.03125, [18] := -1.03125, [19] := -1.03125, [20] := -1.03125, [21] := -1.03125, [22] := -1.03125, [23] := -1.03125, [24] := -1.03125, [25] := -1.03125, [26] := -1.03125, [27] := -1.03125, [28] := -1.03125, [29] := -1.03125);
   FT_1221 : CM_AI_SCL := (RawMin := 4000, RawMax := 20000, EuMax := 48.0, In_Raw := 3993, Percent := -0.04375, PV := -0.021);
   FT_1251 : CM_AI_SCL := (RawMin := 4000, RawMax := 20000, EuMax := 100.0, In_Raw := 3994, Percent := -0.0375, PV := -0.0375);
   FT_202 : CM_AI_SCL := (RawMin := 4000, RawMax := 20000, EuMax := 32571.0, In_Raw := 7539, Percent := 22.11875);
   FT_202_ALT_SCFM : REAL;
   FT_502 : CM_AI_SCL := (RawMin := 4000, RawMax := 20000, EuMax := 32571.0, In_Raw := 7378, Percent := 21.112501);
   FT_502_ALT_SCFM : REAL;
   FT_904 : CM_AI_SCL := (RawMin := 4000, RawMax := 20000, EuMax := 400.0, In_Raw := 4969, Percent := 6.05625);
   FULL_COLLECT_INTERRUPT_ALM : BOOL;
   FULL_COLLECT_INTERRUPT_ALM_TIME : DINT := 30;
   FULL_COLLECT_INTERRUPT_ALM_TMR : TIMER := (PRE := 30000);
   FULL_COLLECT_START_ALM : BOOL;
   FULL_COLLECT_START_ALM_TIME : DINT := 90;
   FULL_COLLECT_START_ALM_TMR : TIMER := (PRE := 90000);
   FVNR550_CommFlt_TON : TIMER := (PRE := 10000, ACC := 27, EN := 1, TT := 1);
   FVNR550_COMMLOSS : BOOL;
   FVNR550_L1Current_HoldingRegister : DINT := 276;
   FVR800C_ChangeDir : BOOL;
   FVR800C_ChangeDirOnStop : BOOL;
   FVR800C_ClearFault_Reset_TMR : TIMER := (PRE := 5000);
   FVR800C_CommFlt_TON : TIMER := (PRE := 10000);
   FVR800C_COMMLOSS : BOOL;
   FVR800C_L1Current_HoldingRegister : DINT;
   FVR800C_RunHours : REAL := 1893.7263;
   FVR800C_RunHoursCTU : COUNTER := (PRE := 8760000, ACC := 1893);
   FVR800C_RunTime : REAL := 1893.0;
   FVR800C_RunTime_CalcHigh : DINT := 2100;
   FVR800C_RunTime_CalcLow : DINT := 2000;
   FVR800C_RunTime_x100Hrs_Current : DINT := 19;
   FVR800C_RunTimer : TIMER := (PRE := 3600000, ACC := 2614851);
   FVR800D_ChangeDir : BOOL;
   FVR800D_ChangeDirOnStop : BOOL;
   FVR800D_ClearFault_Reset_TMR : TIMER := (PRE := 5000);
   FVR800D_CommFlt_TON : TIMER := (PRE := 10000);
   FVR800D_COMMLOSS : BOOL;
   FVR800D_L1Current_HoldingRegister : DINT;
   FVR800D_RunHours : REAL := 1495.5018;
   FVR800D_RunHoursCTU : COUNTER := (PRE := 8760000, ACC := 1495);
   FVR800D_RunTime : REAL := 1495.0;
   FVR800D_RunTime_CalcHigh : DINT := 1700;
   FVR800D_RunTime_CalcLow : DINT := 1600;
   FVR800D_RunTime_x100Hrs_Current : DINT := 15;
   FVR800D_RunTimer : TIMER := (PRE := 3600000, ACC := 1806611);
   FVR_800C_Auto : BOOL := 1;
   FVR_800C_Auto_ONS : BOOL;
   FVR_800C_AutoReq : BOOL;
   FVR_800C_ClearFault_TMR : TIMER := (PRE := 60000);
   FVR_800C_COMMLOSS : BOOL;
   FVR_800C_DISABLE_ONS : BOOL := 1;
   FVR_800C_EN : BOOL;
   FVR_800C_FREQ_OUT : REAL;
   FVR_800C_ManReq : BOOL;
   FVR_800C_ManStartReq : BOOL;
   FVR_800C_PRIMARY : BOOL := 1;
   FVR_800C_RUNNING : BOOL;
   FVR_800C_ST : BOOL;
   FVR_800D_Auto : BOOL := 1;
   FVR_800D_Auto_ONS : BOOL;
   FVR_800D_AutoReq : BOOL;
   FVR_800D_ClearFault_TMR : TIMER;
   FVR_800D_COMMLOSS : BOOL;
   FVR_800D_DISABLE_ONS : BOOL := 1;
   FVR_800D_EN : BOOL;
   FVR_800D_FREQ_OUT : REAL;
   FVR_800D_ManReq : BOOL;
   FVR_800D_ManStartReq : BOOL;
   FVR_800D_PRIMARY : BOOL := 1;
   FVR_800D_RUNNING : BOOL;
   FVR_800D_ST : BOOL;
   Heat_Counter_AT2 : DINT;
   Heat_Counter_AT3 : REAL;
   Heat_Counter_Month : REAL;
   Heat_Counter_Pilot : REAL;
   HEAT_REPORTS : BOOL := 1;
   HEAT_TIMER1 : TIMER := (PRE := 604800000, ACC := 1155655);
   HEAT_TIMER1_MIN : DINT := 19;
   HEAT_TIMER1_MS : DINT := 15655;
   HEAT_TIMER1_SEC : DINT := 15;
   HEAT_TIMER_AT2 : TIMER := (PRE := 604800000, ACC := 1155655);
   HEAT_TIMER_AT2_MIN : DINT := 19;
   HEAT_TIMER_AT2_MS : DINT := 15655;
   HEAT_TIMER_AT2_SEC : DINT := 15;
   HEAT_TIMER_AT3 : TIMER := (PRE := 604800000, ACC := 1259169);
   HEAT_TIMER_AT3_MIN : DINT := 20;
   HEAT_TIMER_AT3_MS : DINT := 59169;
   HEAT_TIMER_AT3_SEC : DINT := 59;
   HEAT_TIMER_PILOT : TIMER := (PRE := 604800000, ACC := 532570);
   HEAT_TIMER_PILOT_MIN : DINT := 8;
   HEAT_TIMER_PILOT_MS : DINT := 52570;
   HEAT_TIMER_PILOT_SEC : DINT := 52;
   HP_Shutoff_PerPump : REAL := 5700.0;
   HP_Shutoff_SPH : DINT := 5100;
   HP_Shutoff_SPL : DINT := 5000;
   HXR_1250 : CM_DO_FVNR := (AlmCurrentHigh_SP := 999.0, Current := -6.25, AlmCD_TmrPre := 5, ProgStartReq := 1, AlmCurrent_TmrPre := 5);
   IGNORE_AT2 : BOOL;   // Ignore all signals from AT2
   IGNORE_AT3 : BOOL;   // Ignore signals from AT3
   IGNORE_TE_802S : BOOL;   // Don't look at TE_802
   IT_1250 : CM_AI_SCL := (RawMin := 4000, RawMax := 20000, EuMax := 100.0, In_Raw := 3000, Percent := -6.25, PV := -6.25);
   LP_SHUTOFF_SPL : REAL := 400.0;
   MANUAL_ARS_LOCKOUT : BOOL;
   MCP_SLOT1_ERROR : BOOL;
   MCP_SLOT2_ERROR : BOOL;
   MCP_SLOT3_ERROR : BOOL;
   MCP_SLOT4_ERROR : BOOL;
   MCP_SLOT5_ERROR : BOOL;
   MODE_ATOMIZE : BOOL;
   MODE_IDLE : BOOL := 1;
   MODE_STANDBY_IDLE : BOOL;
   MODE_STANDBY_PUMPUP : BOOL;
   MODE_STANDBY_RUN : BOOL;
   MTR_200A : CM_DO_FVNR := (AlmCurrentHigh_SP := 999.0, AlmCD_TmrPre := 5, AlmCurrent_TmrPre := 5);
   MTR_550 : CM_DO_FVNR := (Auto := 1, AlmCurrentHigh_SP := 999.0, Current := 2.76, AlmCD_TmrPre := 5, ProgStartReq := 1, Running := 1, Out := 1, AlmCurrent_TmrPre := 5, OperStartReq := 1);
   OFF_TIMER_AT2 : TIMER := (PRE := 10800000, ACC := 10800000, EN := 1, DN := 1);
   OFF_TIMER_AT3 : TIMER := (PRE := 10800000, ACC := 10800000, EN := 1, DN := 1);
   OFF_TIMER_PILOT : TIMER := (PRE := 10800000, ACC := 10800000, EN := 1, DN := 1);
   OLT_1250 : BOOL;   // HXR-1250 Overload Signal
   P_800_COOLDOWN_ALT_TIME : REAL := 900.0;
   P_800_COOLDOWN_ALT_TIME_MS : DINT := 900000;
   P_800A_Cavit : BOOL;
   P_800A_CAVIT_CHK_TMR : TIMER := (PRE := 45000);
   P_800A_CAVIT_CTR : COUNTER := (PRE := 5);
   P_800A_CAVIT_CTR_MONTH : COUNTER := (PRE := 10000);
   P_800A_Cavit_Shutdown : BOOL;
   P_800A_CAVIT_TEMP_SP : DINT := -230;
   P_800A_CAVIT_VENT_START_DLA_TMR : TIMER := (PRE := 5000);
   P_800A_Cavit_Vent_TMR : TIMER := (PRE := 20000);
   P_800A_ClearShutoff : BOOL;
   P_800A_COOLDOWN_ALT_TON : TIMER := (PRE := 900000);
   P_800A_Cooldown_Complete : BOOL;
   P_800A_Direction : BOOL;
   P_800A_Direction_Toggle : BOOL;
   P_800A_Hi_Press_Shutoff : BOOL;
   P_800A_Hi_Press_Vent : BOOL;
   P_800A_Init_OK : BOOL;
   P_800A_Pre_Vent_Done : BOOL;
   P_800A_Pre_Vent_Pending : BOOL;
   P_800A_Prestart : BOOL;
   P_800A_Ready : BOOL;
   P_800A_RUN_OCCURRED : BOOL;
   P_800A_Select_Auto_Online : BOOL;
   P_800A_Start_DLA_TMR : TIMER := (PRE := 60000);
   P_800A_Start_Temp_SP : DINT := -270;
   P_800A_Start_TMR : TIMER := (PRE := 2000);
   P_800A_Start_Vent_TMR : TIMER := (PRE := 45000);
   P_800A_STOP_ONS : BOOL;
   P_800A_Stop_Vent_Delay : BOOL;
   P_800A_Stop_Vent_TMR : TIMER := (PRE := 20000);
   P_800B_Cavit : BOOL;
   P_800B_CAVIT_CHK_TMR : TIMER := (PRE := 45000);
   P_800B_CAVIT_CTR : COUNTER := (PRE := 5);
   P_800B_CAVIT_CTR_MONTH : COUNTER := (PRE := 10000);
   P_800B_Cavit_Shutdown : BOOL;
   P_800B_CAVIT_TEMP_SP : DINT := -230;
   P_800B_CAVIT_VENT_START_DLA_TMR : TIMER := (PRE := 5000);
   P_800B_Cavit_Vent_TMR : TIMER := (PRE := 20000);
   P_800B_ClearShutoff : BOOL;
   P_800B_COOLDOWN_ALT_TON : TIMER := (PRE := 900000);
   P_800B_Cooldown_Complete : BOOL;
   P_800B_Direction : BOOL;
   P_800B_Direction_Toggle : BOOL;
   P_800B_Hi_Press_Shutoff : BOOL;
   P_800B_Hi_Press_Vent : BOOL;
   P_800B_Init_OK : BOOL;
   P_800B_Pre_Vent_Done : BOOL;
   P_800B_Pre_Vent_Pending : BOOL;
   P_800B_Prestart : BOOL;
   P_800B_Ready : BOOL;
   P_800B_RUN_OCCURRED : BOOL;
   P_800B_Select_Auto_Online : BOOL;
   P_800B_Start_DLA_TMR : TIMER := (PRE := 60000);
   P_800B_Start_Temp_SP : DINT := -270;
   P_800B_Start_TMR : TIMER := (PRE := 2000);
   P_800B_Start_Vent_TMR : TIMER := (PRE := 45000);
   P_800B_STOP_ONS : BOOL;
   P_800B_Stop_Vent_Delay : BOOL;
   P_800B_Stop_Vent_TMR : TIMER := (PRE := 20000);
   P_800C : CM_DO_FVR := (Auto := 1, AlmCurrentHigh_SP := 999.0, AlmCD_TmrPre := 5, AlmCurrent_TmrPre := 5);
   P_800C_Cavit : BOOL;
   P_800C_CAVIT_CHK_TMR : TIMER := (PRE := 45000);
   P_800C_CAVIT_CTR : COUNTER := (PRE := 5);
   P_800C_CAVIT_CTR_MONTH : COUNTER := (PRE := 10000);
   P_800C_Cavit_Shutdown : BOOL;
   P_800C_CAVIT_TEMP_SP : DINT := -230;
   P_800C_CAVIT_VENT_START_DLA_TMR : TIMER := (PRE := 5000);
   P_800C_Cavit_Vent_TMR : TIMER := (PRE := 20000);
   P_800C_ClearShutoff : BOOL;
   P_800C_COOLDOWN_ALT_TON : TIMER := (PRE := 900000);
   P_800C_Cooldown_Complete : BOOL;
   P_800C_Direction : BOOL;
   P_800C_Direction_Toggle : BOOL;
   P_800C_EN : BOOL;
   P_800C_Fault : BOOL;
   P_800C_Hi_Press_Shutoff : BOOL;
   P_800C_Hi_Press_Vent : BOOL;
   P_800C_Init_OK : BOOL;
   P_800C_Pre_Vent_Done : BOOL;
   P_800C_Pre_Vent_Pending : BOOL;
   P_800C_Prestart : BOOL;
   P_800C_Ready : BOOL;
   P_800C_RUN_OCCURRED : BOOL;
   P_800C_Select_Auto_Online : BOOL;
   P_800C_ST : BOOL;
   P_800C_Start_DLA_TMR : TIMER := (PRE := 60000);
   P_800C_Start_Temp_SP : DINT := -270;
   P_800C_Start_TMR : TIMER := (PRE := 2000);
   P_800C_Start_Vent_TMR : TIMER := (PRE := 45000);
   P_800C_STOP_ONS : BOOL;
   P_800C_Stop_Vent_Delay : BOOL;
   P_800C_Stop_Vent_TMR : TIMER := (PRE := 20000);
   P_800D : CM_DO_FVR := (Auto := 1, AlmCurrentHigh_SP := 999.0, AlmCD_TmrPre := 5, AlmCurrent_TmrPre := 5);
   P_800D_Cavit : BOOL;
   P_800D_CAVIT_CHK_TMR : TIMER := (PRE := 45000);
   P_800D_CAVIT_CTR : COUNTER := (PRE := 5);
   P_800D_CAVIT_CTR_MONTH : COUNTER := (PRE := 10000);
   P_800D_Cavit_Shutdown : BOOL;
   P_800D_CAVIT_TEMP_SP : DINT := -230;
   P_800D_CAVIT_VENT_START_DLA_TMR : TIMER := (PRE := 5000);
   P_800D_Cavit_Vent_TMR : TIMER := (PRE := 20000);
   P_800D_ClearShutoff : BOOL;
   P_800D_COOLDOWN_ALT_TON : TIMER := (PRE := 900000);
   P_800D_Cooldown_Complete : BOOL;
   P_800D_Direction : BOOL;
   P_800D_Direction_Toggle : BOOL;
   P_800D_EN : BOOL;
   P_800D_Fault : BOOL;
   P_800D_Hi_Press_Shutoff : BOOL;
   P_800D_Hi_Press_Vent : BOOL;
   P_800D_Init_OK : BOOL;
   P_800D_Pre_Vent_Done : BOOL;
   P_800D_Pre_Vent_Pending : BOOL;
   P_800D_Prestart : BOOL;
   P_800D_Ready : BOOL;
   P_800D_RUN_OCCURRED : BOOL;
   P_800D_Select_Auto_Online : BOOL;
   P_800D_ST : BOOL;
   P_800D_Start_DLA_TMR : TIMER := (PRE := 60000);
   P_800D_Start_Temp_SP : DINT := -270;
   P_800D_Start_TMR : TIMER := (PRE := 2000);
   P_800D_Start_Vent_TMR : TIMER := (PRE := 45000);
   P_800D_STOP_ONS : BOOL;
   P_800D_Stop_Vent_Delay : BOOL;
   P_800D_Stop_Vent_TMR : TIMER := (PRE := 20000);
   PDT_1101A : CM_AI_SCL_ALT := (RawMin := 4000, RawMax := 20000, EuMax := 45.0, AltScaleMultiplier := 27.7, In_Raw := 7192, Percent := 19.949999, PV := 8.9775, AltScalePV := 248.67676);
   PDT_1301A : CM_AI_SCL_ALT := (RawMin := 4000, RawMax := 20000, EuMax := 45.0, AltScaleMultiplier := 27.7, In_Raw := 7467, Percent := 21.66875, PV := 9.750937, AltScalePV := 270.10098);
   PDT_1301B : CM_AI_SCL_ALT := (RawMin := 4000, RawMax := 20000, EuMax := 45.0, AltScaleMultiplier := 27.7, In_Raw := 7283, Percent := 20.51875, PV := 9.233438, AltScalePV := 255.76622);
   PDT_601 : CM_AI_SCL_ALT := (RawMin := 4000, RawMax := 20000, EuMax := 45.0, AltScaleMultiplier := 27.7, In_Raw := 3994, Percent := -0.0375, PV := -0.016875, AltScalePV := -0.46743754);
   PDT_603 : CM_AI_SCL_ALT := (RawMin := 4000, RawMax := 20000, EuMax := 15.0, AltScaleMultiplier := 27.7, In_Raw := 3993, Percent := -0.04375, PV := -0.0065625, AltScalePV := -0.18178125);
   PDT_603_PERCENT : REAL := -0.10195247;
   PDT_701 : CM_AI_SCL_ALT := (RawMin := 4000, RawMax := 20000, EuMax := 45.0, AltScaleMultiplier := 27.7, In_Raw := 3993, Percent := -0.04375, PV := -0.0196875, AltScalePV := -0.54534376);
   PDT_701_ALT_GAL : REAL := -3.9517572;
   PDT_701_ALT_SCF : REAL := -444.3751;
   PDT_721_CALC : REAL := -0.30862466;
   PDT_751 : CM_AI_SCL_ALT := (RawMin := 4000, RawMax := 20000, EuMax := 15.0, AltScaleMultiplier := 27.7, In_Raw := 3990, Percent := -0.06250001, PV := -0.009375, AltScalePV := -0.2596875);
   PDT_753 : CM_AI_SCL_ALT := (RawMin := 4000, RawMax := 20000, EuMax := 15.0, AltScaleMultiplier := 27.7, In_Raw := 3990, Percent := -0.06250001, PV := -0.009375, AltScalePV := -0.2596875);
   PDT_851_InRange : BOOL;
   PIDE_1001 : PID_ENHANCED := (PV := 2392.3188, PVEUMax := 6700.0, SPProg := 2450.0, SPOper := 2450.0, SPHLimit := 4000.0, RatioProg := 1.0, RatioOper := 1.0, RatioHLimit := 1.0, RatioLLimit := 1.0, CVProg := 20.0, CVOper := 100.0, CVEUMax := 100.0, CVHLimit := 100.0, DependIndepend := 1, PGain := 8.0, IGain := 0.2, PVEDerivative := 1, ProgAutoReq := 1, RTSTime := 1, CVEU := 100.0, CV := 100.0, CVHAlarm := 1, SP := 2450.0, SPPercent := 36.56716, PVPercent := 35.706253, E := 57.681152, EPercent := 0.8609085, InitPrimary := 1, WindupHOut := 1, Ratio := 1.0, ProgOper := 1, Auto := 1, DeltaT := 0.1);
   PIDE_1002 : PID_ENHANCED := (PV := 2230.875, PVEUMax := 3000.0, SPProg := 2350.0, SPOper := 2350.0, SPHLimit := 3000.0, RatioProg := 1.0, RatioOper := 1.0, RatioHLimit := 1.0, RatioLLimit := 1.0, CVOper := 30.0, CVEUMax := 100.0, CVHLimit := 80.0, CVROCLimit := 4.0, DependIndepend := 1, PGain := 6.0, IGain := 0.2, PVEDerivative := 1, ProgAutoReq := 1, RTSTime := 1, CVEU := 30.0, CV := 30.0, SP := 2350.0, SPPercent := 78.333336, PVPercent := 74.362495, E := 119.125, EPercent := 3.9708405, InitPrimary := 1, Ratio := 1.0, Manual := 1, DeltaT := 0.1);
   PIDE_1002_FLOW_IGAIN : REAL := 0.07;
   PIDE_1002_FLOW_PGAIN : REAL := 0.2;
   PIDE_1002_FLOW_SP : PID_ENHANCED := (PV := 5.6725345, PVEUMax := 1000.0, SPHLimit := 200.0, RatioProg := 1.0, RatioOper := 1.0, RatioHLimit := 1.0, RatioLLimit := 1.0, CVEUMax := 126.03422, CVHLimit := 100.0, PGain := 1.0, IGain := 0.5, PVEDerivative := 1, ProgManualReq := 1, RTSTime := 1, PVPercent := 0.5672535, E := -5.6725345, EPercent := -0.5672535, InitPrimary := 1, Ratio := 1.0, Manual := 1, DeltaT := 0.1);
   PIDE_1002_PRESSURE_IGAIN : REAL := 0.2;
   PIDE_1002_PRESSURE_PGAIN : REAL := 6.0;
   PIDE_1002_PVCHANGE0 : BOOL := 1;
   PIDE_1002_PVCHANGE1 : BOOL;
   PIDE_1002_RESET : BOOL := 1;
   PIDE_1003 : PID_ENHANCED := (PVEUMax := 100.0, SPHLimit := 100.0, RatioProg := 1.0, RatioOper := 1.0, RatioHLimit := 1.0, RatioLLimit := 1.0, CVEUMax := 100.0, CVHLimit := 100.0, PVEDerivative := 1, RTSTime := 1);
   PIDE_101A : PID_ENHANCED := (PV := 1.4749999, PVEUMax := 5.0, PVEUMin := -5.0, SPProg := 0.1, SPOper := 0.1, SPHLimit := 5.0, RatioProg := 1.0, RatioOper := 1.0, RatioHLimit := 1.0, RatioLLimit := 1.0, CVEUMax := 100.0, CVHLimit := 100.0, CVROCLimit := 5.0, ControlAction := 1, DependIndepend := 1, PGain := 5.0, IGain := 0.5, PVEDerivative := 1, ProgManualReq := 1, RTSTime := 1, SP := 0.1, SPPercent := 51.0, PVPercent := 64.75, E := 1.3749999, EPercent := 13.75, InitPrimary := 1, Ratio := 1.0, ProgOper := 1, Manual := 1, DeltaT := 0.1);
   PIDE_101B : PID_ENHANCED := (PV := 0.6574998, PVEUMax := 5.0, PVEUMin := -5.0, SPHLimit := 5.0, RatioProg := 1.0, RatioOper := 1.0, RatioHLimit := 1.0, RatioLLimit := 1.0, CVEUMax := 100.0, CVHLimit := 100.0, ControlAction := 1, DependIndepend := 1, PGain := 3.0, IGain := 0.5, PVEDerivative := 1, ProgManualReq := 1, RTSTime := 1, SPPercent := 50.0, PVPercent := 56.575, E := 0.6574998, EPercent := 6.575001, InitPrimary := 1, Ratio := 1.0, ProgOper := 1, Manual := 1, DeltaT := 0.1);
   PIDE_101C : PID_ENHANCED := (PV := 1.674375, PVEUMax := 5.0, PVEUMin := -5.0, SPHLimit := 5.0, RatioProg := 1.0, RatioOper := 1.0, RatioHLimit := 1.0, RatioLLimit := 1.0, CVEUMax := 100.0, CVHLimit := 100.0, ControlAction := 1, DependIndepend := 1, PGain := 3.0, IGain := 0.5, PVEDerivative := 1, ProgManualReq := 1, RTSTime := 1, SPPercent := 50.0, PVPercent := 66.74375, E := 1.674375, EPercent := 16.743752, InitPrimary := 1, Ratio := 1.0, ProgOper := 1, Manual := 1, DeltaT := 0.1);
   PIDE_102A : PID_ENHANCED := (PV := 1.5193748, PVEUMax := 5.0, PVEUMin := -5.0, SPProg := 1.5, SPOper := 1.5, SPHLimit := 5.0, RatioProg := 1.0, RatioOper := 1.0, RatioHLimit := 1.0, RatioLLimit := 1.0, CVProg := 50.0, CVOper := 2.3181522, CVEUMax := 100.0, CVHLimit := 100.0, CVROCLimit := 7.0, ControlAction := 1, DependIndepend := 1, PGain := 4.0, IGain := 0.5, PVEDerivative := 1, ProgAutoReq := 1, RTSTime := 1, CVEU := 2.3181522, CV := 2.3181522, SP := 1.5, SPPercent := 65.0, PVPercent := 65.19375, E := 0.019374847, EPercent := 0.19374847, InitPrimary := 1, Ratio := 1.0, ProgOper := 1, Auto := 1, DeltaT := 0.1);
   PIDE_102B : PID_ENHANCED := (PV := 0.64125013, PVEUMax := 5.0, PVEUMin := -5.0, SPProg := 1.5, SPOper := 1.5, SPHLimit := 5.0, RatioProg := 1.0, RatioOper := 1.0, RatioHLimit := 1.0, RatioLLimit := 1.0, CVProg := 50.0, CVOper := 4.0, CVEUMax := 100.0, CVHLimit := 100.0, CVLLimit := 4.0, ControlAction := 1, DependIndepend := 1, PGain := 3.0, IGain := 0.5, PVEDerivative := 1, ProgAutoReq := 1, RTSTime := 1, CVEU := 4.0, CV := 4.0, CVLAlarm := 1, SP := 1.5, SPPercent := 65.0, PVPercent := 56.4125, E := -0.85874987, EPercent := -8.587502, InitPrimary := 1, WindupHOut := 1, Ratio := 1.0, ProgOper := 1, Auto := 1, DeltaT := 0.1);
   PIDE_102C : PID_ENHANCED := (PV := 1.21, PVEUMax := 5.0, PVEUMin := -5.0, SPProg := 1.5, SPOper := 1.5, SPHLimit := 5.0, RatioProg := 1.0, RatioOper := 1.0, RatioHLimit := 1.0, RatioLLimit := 1.0, CVProg := 50.0, CVOper := 0.010931406, CVEUMax := 100.0, CVHLimit := 100.0, ControlAction := 1, DependIndepend := 1, PGain := 3.0, IGain := 0.5, PVEDerivative := 1, ProgAutoReq := 1, RTSTime := 1, CVEU := 0.010931406, CV := 0.010931406, SP := 1.5, SPPercent := 65.0, PVPercent := 62.1, E := -0.28999996, EPercent := -2.9000015, InitPrimary := 1, Ratio := 1.0, ProgOper := 1, Auto := 1, DeltaT := 0.1);
   PIDE_1221 : PID_ENHANCED := (PV := -0.021, PVEUMax := 48.0, SPProg := 1.0, SPOper := 1.0, SPHLimit := 3.0, RatioProg := 1.0, RatioOper := 1.0, RatioHLimit := 1.0, RatioLLimit := 1.0, CVEUMax := 100.0, CVHLimit := 100.0, DependIndepend := 1, PGain := 2.0, IGain := 0.1, PVEDerivative := 1, ProgManualReq := 1, RTSTime := 1, SP := 1.0, SPPercent := 2.0833335, PVPercent := -0.04375, E := 1.021, EPercent := 2.1270835, InitPrimary := 1, Ratio := 1.0, Manual := 1, DeltaT := 0.1);
   PIDE_1251 : PID_ENHANCED := (PV := -0.0375, PVEUMax := 100.0, SPProg := 30.0, SPOper := 30.0, SPHLimit := 100.0, RatioProg := 1.0, RatioOper := 1.0, RatioHLimit := 1.0, RatioLLimit := 1.0, CVEUMax := 100.0, CVHLimit := 100.0, DependIndepend := 1, PGain := 2.0, IGain := 0.1, PVEDerivative := 1, ProgManualReq := 1, RTSTime := 1, SP := 30.0, SPPercent := 30.000002, PVPercent := -0.0375, E := 30.0375, EPercent := 30.037502, InitPrimary := 1, Ratio := 1.0, Manual := 1, DeltaT := 0.1);
   PIDE_202 : PID_ENHANCED := (PV := 1.3868752, PVEUMax := 5.0, PVEUMin := -5.0, SPProg := 0.4, SPOper := 0.4, SPHLimit := 5.0, RatioProg := 1.0, RatioOper := 1.0, RatioHLimit := 1.0, RatioLLimit := 1.0, CVEUMax := 100.0, CVHLimit := 100.0, CVROCLimit := 3.0, ControlAction := 1, DependIndepend := 1, PGain := 5.0, IGain := 0.55, PVEDerivative := 1, ProgManualReq := 1, RTSTime := 1, SP := 0.4, SPPercent := 54.000004, PVPercent := 63.868748, E := 0.9868752, EPercent := 9.868744, InitPrimary := 1, Ratio := 1.0, ProgOper := 1, Manual := 1, DeltaT := 0.1);
   PIDE_204 : PID_ENHANCED := (PV := 1.3987498, PVEUMax := 5.0, PVEUMin := -5.0, SPProg := 1.6, SPOper := 1.6, SPHLimit := 5.0, RatioProg := 1.0, RatioOper := 1.0, RatioHLimit := 1.0, RatioLLimit := 1.0, CVProg := 40.0, CVEUMax := 100.0, CVHLimit := 100.0, CVROCLimit := 5.0, ControlAction := 1, DependIndepend := 1, PGain := 2.5, IGain := 0.4, PVEDerivative := 1, ProgAutoReq := 1, RTSTime := 1, CVLAlarm := 1, SP := 1.6, SPPercent := 66.0, PVPercent := 63.9875, E := -0.2012502, EPercent := -2.0125008, InitPrimary := 1, WindupHOut := 1, Ratio := 1.0, ProgOper := 1, Auto := 1, DeltaT := 0.1);
   PIDE_207 : PID_ENHANCED := (PV := 3.474701, PVEUMax := 145.0, PVEUMin := -14.6, SPProg := 0.2, SPOper := 0.2, SPHLimit := 100.0, RatioProg := 1.0, RatioOper := 1.0, RatioHLimit := 1.0, RatioLLimit := 1.0, CVEUMax := 100.0, CVHLimit := 100.0, DependIndepend := 1, PGain := 2.0, IGain := 0.5, PVEDerivative := 1, ProgManualReq := 1, RTSTime := 1, SP := 0.2, SPPercent := 9.273183, PVPercent := 11.325, E := -3.2747009, EPercent := -2.051817, InitPrimary := 1, Ratio := 1.0, Manual := 1, DeltaT := 0.1);
   PIDE_207_RECYCLE : BOOL;
   PIDE_207_SP_PT1002 : REAL := 1350.0;
   PIDE_207_SP_PT601 : REAL := 2.0;
   PIDE_504 : PID_ENHANCED := (PV := 56.801056, PVEUMax := 145.0, PVEUMin := -14.6, SPProg := 50.0, SPOper := 50.0, SPHLimit := 100.0, SPLLimit := -2.0, RatioProg := 1.0, RatioOper := 1.0, RatioHLimit := 1.0, RatioLLimit := 1.0, CVProg := 50.0, CVOper := 10.0, CVEUMax := 100.0, CVHLimit := 100.0, ControlAction := 1, DependIndepend := 1, PGain := 13.0, IGain := 0.24, PVEDerivative := 1, ProgAutoReq := 1, RTSTime := 1, CVEU := 10.0, CV := 10.0, SP := 50.0, SPPercent := 40.47619, PVPercent := 44.7375, E := 6.801056, EPercent := 4.2613106, InitPrimary := 1, Ratio := 1.0, Manual := 1, DeltaT := 0.1);
   PIDE_504_COLDBOX_IGAIN : REAL := 0.24;
   PIDE_504_COLDBOX_PGAIN : REAL := 13.0;
   PIDE_504_FRONT_END_CONTROL : BOOL;
   PIDE_504_FRONT_END_CONTROL_REQUEST : BOOL := 1;
   PIDE_504_FRONT_END_IGAIN : REAL := 0.2;
   PIDE_504_FRONT_END_PGAIN : REAL := 3.0;
   PIDE_504_MODE : BOOL := 1;   // 0 = Argon (PT-601) 1 = N2 (PT-603)
   PIDE_504_PVCHANGE1 : BOOL;
   PIDE_504_PVCHANGE2 : BOOL := 1;
   PIDE_504_PVCHANGE3 : BOOL;
   PIDE_504_RESET : BOOL := 1;
   PIDE_603 : PID_ENHANCED := (PV := -0.18178125, PVEUMax := 1246.5, SPProg := 120.0, SPOper := 120.0, SPHLimit := 186.0, RatioProg := 1.0, RatioOper := 1.0, RatioHLimit := 1.0, RatioLLimit := 1.0, CVProg := 60.0, CVOper := 60.0, CVEUMax := 100.0, CVHLimit := 100.0, DependIndepend := 1, PGain := 10.0, IGain := 0.5, PVEDerivative := 1, ProgAutoReq := 1, RTSTime := 1, CVEU := 60.0, CV := 60.0, SP := 120.0, SPPercent := 9.626956, PVPercent := -0.014583332, E := 120.18178, EPercent := 9.64154, InitPrimary := 1, Ratio := 1.0, Manual := 1, DeltaT := 0.1);
   PIDE_603_CVLimit_TON : TIMER := (PRE := 5000);
   PIDE_603_CVLimitLOW_TON : TIMER := (PRE := 5000);
   PIDE_605 : PID_ENHANCED := (PV := 2.9460258, PVEUMax := 145.0, PVEUMin := -14.6, SPProg := 7.0, SPOper := 7.0, SPHLimit := 100.0, RatioProg := 1.0, RatioOper := 1.0, RatioHLimit := 1.0, RatioLLimit := 1.0, CVEUMax := 100.0, CVHLimit := 100.0, ControlAction := 1, DependIndepend := 1, PGain := 3.5, IGain := 0.01, PVEDerivative := 1, ProgAutoReq := 1, RTSTime := 1, CVLAlarm := 1, SP := 7.0, SPPercent := 13.5338335, PVPercent := 10.993751, E := -4.053974, EPercent := -2.540083, InitPrimary := 1, WindupHOut := 1, Ratio := 1.0, ProgOper := 1, Auto := 1, DeltaT := 0.1);
   PIDE_753 : PID_ENHANCED := (PV := -0.28565627, PVEUMax := 415.5, SPProg := 4.0, SPOper := 4.0, SPHLimit := 25.0, RatioProg := 1.0, RatioOper := 1.0, RatioHLimit := 1.0, RatioLLimit := 1.0, CVEUMax := 100.0, CVHLimit := 20.0, DependIndepend := 1, PGain := 3.5, IGain := 0.05, PVEDerivative := 1, ProgAutoReq := 1, RTSTime := 1, SP := 4.0, SPPercent := 0.9626956, PVPercent := -0.06875001, E := 4.2856565, EPercent := 1.0314456, InitPrimary := 1, Ratio := 1.0, Manual := 1, DeltaT := 0.1);
   PIDE_754 : PID_ENHANCED := (PV := -15.467825, PVEUMax := 145.0, PVEUMin := -14.6, SPProg := 24.0, SPOper := 70.0, SPHLimit := 100.0, RatioProg := 1.0, RatioOper := 1.0, RatioHLimit := 1.0, RatioLLimit := 1.0, CVEUMax := 100.0, CVHLimit := 50.0, ControlAction := 1, DependIndepend := 1, PGain := 10.0, IGain := 0.8, PVEDerivative := 1, ProgAutoReq := 1, RTSTime := 1, SP := 70.0, SPPercent := 53.007515, PVPercent := -0.5437497, E := -85.46783, EPercent := -53.551266, InitPrimary := 1, Ratio := 1.0, Manual := 1, DeltaT := 0.1);
   PIDE_755 : PID_ENHANCED := (PV := -0.2596875, PVEUMax := 415.5, SPProg := 82.0, SPOper := 82.0, SPHLimit := 100.0, RatioProg := 1.0, RatioOper := 1.0, RatioHLimit := 1.0, RatioLLimit := 1.0, CVEUMax := 100.0, CVHLimit := 100.0, DependIndepend := 1, PGain := 3.0, IGain := 0.1, PVEDerivative := 1, ProgManualReq := 1, RTSTime := 1, SP := 82.0, SPPercent := 19.735258, PVPercent := -0.06250001, E := 82.25969, EPercent := 19.797758, InitPrimary := 1, Ratio := 1.0, ProgOper := 1, Manual := 1, DeltaT := 0.1);
   PIDE_800 : PID_ENHANCED := (PV := 2394.8313, PVEUMax := 6700.0, SPProg := 4800.0, SPOper := 4800.0, SPHLimit := 5800.0, RatioProg := 1.0, RatioOper := 1.0, RatioHLimit := 1.0, RatioLLimit := 1.0, CVProg := 100.0, CVOper := 100.0, CVManLimiting := 1, CVEUMax := 60.0, CVHLimit := 100.0, CVLLimit := 33.0, CVROCLimit := 20.0, DependIndepend := 1, PGain := 6.0, IGain := 3.0, ProgManualReq := 1, RTSTime := 1, CVEU := 60.0, CV := 100.0, SP := 4800.0, SPPercent := 71.64179, PVPercent := 35.74375, E := 2405.1687, EPercent := 35.89804, InitPrimary := 1, Ratio := 1.0, ProgOper := 1, Manual := 1, DeltaT := 0.1);
   PIDE_800_CVOper_HZ : REAL := 60.0;
   PIDE_800_CVProg_HZ : REAL := 60.0;
   PIDE_800_InRange : BOOL;
   PIDE_800_OPER_ONS : BOOL;
   PILOT_ATOMIZE_FLOW : REAL;
   PILOT_ATOMIZE_VALVE_OPEN : BOOL;   // Halo Valve
   Pilot_Atomizing_Valve_Close_TON : TIMER := (PRE := 30000, ACC := 30000, EN := 1, DN := 1);
   Pilot_Atomizing_Valve_Open_TON : TIMER := (PRE := 5000);
   Pilot_AtomizingStatus_OSF_OB : BOOL;
   Pilot_AtomizingStatus_OSF_SB : BOOL;
   Pilot_AtomizingStatus_OSR_OB : BOOL;
   Pilot_AtomizingStatus_OSR_SB : BOOL;
   PILOT_COMM_STATUS : BOOL := 1;
   PILOT_EXHAUST_VALVE_OPEN : BOOL;
   PILOT_FT_202_TOTAL_HEAT : REAL;
   PILOT_INLET_FLOW : REAL;
   PILOT_INLET_VALVE_OPEN : BOOL;   // Pressure Control Status (Backfill)
   Pilot_Inlet_Valve_Open_TON : TIMER := (PRE := 2000);
   PILOT_MELT_STATUS : BOOL;
   PILOT_PARTICULATE_POST_FILTER : REAL;
   PILOT_PEDESTAL_LEVEL : REAL;
   PILOT_PLANT_ATOMIZING : BOOL;
   PILOT_PLANT_ATOMIZING_ONS : BOOL;
   PILOT_PLANT_BACKFILL : BOOL;
   PILOT_PLANT_BACKFILL_COOLDOWN_DLA : REAL;
   PILOT_PLANT_BACKFILL_COOLDOWN_DLA_SEC : REAL := 3000.0;
   PILOT_PLANT_BACKFILL_COOLDOWN_DLA_TMR : TIMER := (PRE := 3000000);   // delays the cooldown for a backfill
   PILOT_PLANT_BACKFILL_TIMEOUT_TMR : TIMER := (PRE := 1800000);
   PILOT_PLANT_COLLECT_AUTO : BOOL;
   PILOT_PLANT_COLLECTING : BOOL;
   PILOT_PLANT_COLLECTION_PERCENT : REAL := 56.70907;
   PILOT_PLANT_COLLECTION_PERCENT_GOOD_GAS : REAL := 76.501915;
   PILOT_PLANT_COLLECTION_TIME : TIMER := (PRE := 6000000, ACC := 288465);
   PILOT_PLANT_COMMLOSS : BOOL;
   PILOT_PLANT_GOOD_GAS_PERCENT : REAL := 70.80177;
   PILOT_PLANT_GOOD_GAS_TIME : TIMER := (PRE := 7200000, ACC := 377069);   // PILOT time with good gas and no collection stops
   PILOT_PLANT_GOOD_H2O_PERCENT : REAL := 98.122314;
   PILOT_PLANT_GOOD_H2O_TIME : TIMER := (PRE := 7200000, ACC := 522570);   // PILOT time with good dew point and no collection stop
   PILOT_PLANT_GOOD_O2_PERCENT : REAL := 70.80177;
   PILOT_PLANT_GOOD_O2_TIME : TIMER := (PRE := 7200000, ACC := 377069);   // PILOT time with good O2 and no collection stop
   PILOT_PLANT_H2O_MIN : REAL := -82.365;   // Pilot Heat Minimum after burp
   PILOT_PLANT_LIKELY_COLLECTING : BOOL;
   PILOT_PLANT_LIKELY_COLLECTION_TIME : TIMER := (PRE := 6000000, ACC := 315566);
   PILOT_PLANT_MAX_H2O : REAL := -81.686874;
   PILOT_PLANT_MAX_O2 : REAL := 74.5;
   PILOT_PLANT_O2_MIN : REAL := 4.5;   // Pilot Heat Minimum after burp
   PILOT_PLANT_POST_ATOMIZING_TON : TIMER := (PRE := 1200000, ACC := 1200000, EN := 1, DN := 1);
   PILOT_PLANT_POST_HEAT_NOTIFICATION_TON : TIMER := (PRE := 10000, ACC := 10000, EN := 1, DN := 1);
   PILOT_PLANT_RETURN_AUTO : BOOL := 1;
   PILOT_PT_101A_Pressure_Override : REAL := 3.0;   // Pressure at which 101A will be allowed despite any control limitations, intended as a rescue setpoint, not an interlock
   PK_TEST : BOOL;
   PLC_S1_TOF : TIMER := (PRE := 1000, ACC := 1000);
   PLC_S2_TOF : TIMER := (PRE := 1000, ACC := 1000);
   PLC_S3_TOF : TIMER := (PRE := 1000, ACC := 1000);
   PLC_S4_TOF : TIMER := (PRE := 1000, ACC := 1000);
   PLC_S5_TOF : TIMER := (PRE := 1000, ACC := 1000);
   PRAX_N2_ASSUME : REAL := 5.0;
   PT_051 : CM_AI_SCL := (RawMin := 4000, RawMax := 20000, EuMin := -14.6, EuMax := 145.0, In_Raw := 14729, Percent := 63.739162, PV := 92.42178);
   PT_1001 : CM_AI_SCL := (RawMin := 4000, RawMax := 20000, EuMax := 6700.0, In_Raw := 9713, Percent := 35.706253, PV := 2392.3188);
   PT_1001_MINUS_10 : REAL := 2382.3188;
   PT_1001_MINUS_50 : REAL := 2342.3188;
   PT_1002 : CM_AI_SCL := (RawMin := 4000, RawMax := 20000, EuMax := 3625.0, In_Raw := 13660, Percent := 60.375, PV := 2188.5938);
   PT_1003 : CM_AI_SCL := (RawMin := 4000, RawMax := 20000, EuMax := 3000.0, In_Raw := 15907, Percent := 74.41875, PV := 2232.5625);
   PT_101A : CM_AI_SCL := (RawMin := 4000, RawMax := 20000, EuMin := -5.0, EuMax := 5.0, In_Raw := 14353, Percent := 29.412498, PV := 1.4706249);
   PT_101B : CM_AI_SCL := (RawMin := 4000, RawMax := 20000, EuMin := -5.0, EuMax := 5.0, In_Raw := 13021, Percent := 12.762499, PV := 0.63812494);
   PT_101B_SPH : REAL := 0.1;
   PT_101B_SPL : REAL;
   PT_101C : CM_AI_SCL := (RawMin := 4000, RawMax := 20000, EuMin := -5.0, EuMax := 5.0, In_Raw := 14386, Percent := 29.825003, PV := 1.49125);
   PT_101C_SPH : REAL := 0.6;
   PT_101C_SPL : REAL;
   PT_1101A : CM_AI_SCL := (RawMin := 4000, RawMax := 20000, EuMax := 150.0, In_Raw := 8392, Percent := 27.449999, PV := 41.175);
   PT_1201 : CM_AI_SCL := (RawMin := 4000, RawMax := 20000, EuMax := 3000.0, In_Raw := 16945, Percent := 80.90625, PV := 2427.1875);
   PT_1220 : CM_AI_SCL := (RawMin := 4000, RawMax := 20000, EuMax := 3000.0, In_Raw := 3948, Percent := -0.32500002, PV := -9.75);
   PT_1222 : CM_AI_SCL := (RawMin := 4000, RawMax := 20000, EuMax := 150.0, In_Raw := 4070, Percent := 0.4375, PV := 0.65625);
   PT_1301A : CM_AI_SCL := (RawMin := 4000, RawMax := 20000, EuMax := 150.0, In_Raw := 9098, Percent := 31.862501, PV := 47.79375);
   PT_1301B : CM_AI_SCL := (RawMin := 4000, RawMax := 20000, EuMax := 150.0, In_Raw := 9040, Percent := 31.5, PV := 47.25);
   PT_201 : CM_AI_SCL := (RawMin := 4000, RawMax := 20000, EuMin := -5.0, EuMax := 5.0, In_Raw := 14219, Percent := 27.737505, PV := 1.3868752);
   PT_222 : CM_AI_SCL := (RawMin := 4000, RawMax := 20000, EuMin := -14.6, EuMax := 145.0, In_Raw := 13231, Percent := 53.43395, PV := 77.479225);
   PT_601 : CM_AI_SCL := (RawMin := 4000, RawMax := 20000, EuMin := -14.6, EuMax := 145.0, In_Raw := 5695, Percent := 1.5914655, PV := 2.3076248);
   PT_601_FCV_202_SP : REAL := 2.0;
   PT_601_LR : CM_AI_SCL := (RawMin := 4000, RawMax := 20000, EuMin := -14.5, EuMax := 14.5, In_Raw := 13388, Percent := 17.350006, PV := 2.515751);
   PT_603 : CM_AI_SCL := (RawMin := 4000, RawMax := 20000, EuMin := -14.6, EuMax := 145.0, In_Raw := 11141, Percent := 39.05619, PV := 56.631477);
   PT_701 : CM_AI_SCL := (RawMin := 4000, RawMax := 20000, EuMin := -14.6, EuMax := 145.0, In_Raw := 5759, Percent := 2.031742, PV := 2.9460258);
   PT_721 : CM_AI_SCL := (RawMin := 4000, RawMax := 20000, EuMin := -14.6, EuMax := 145.0, In_Raw := 5716, Percent := 1.735932, PV := 2.5171013);
   PT_751 : CM_AI_SCL := (RawMin := 4000, RawMax := 20000, EuMin := -14.6, EuMax := 145.0, In_Raw := 5874, Percent := 2.8228614, PV := 4.093149);
   PT_753 : CM_AI_SCL := (RawMin := 4000, RawMax := 20000, EuMin := -14.6, EuMax := 145.0, In_Raw := 3913, Percent := -10.667465, PV := -15.467825);
   PT_802A : CM_AI_SCL := (RawMin := 4000, RawMax := 20000, EuMax := 6700.0, In_Raw := 4000);
   PT_802B : CM_AI_SCL := (RawMin := 4000, RawMax := 20000, EuMax := 8702.0, In_Raw := 3999, Percent := -0.0062499996, PV := -0.543875);
   PT_802C : CM_AI_SCL := (RawMin := 4000, RawMax := 20000, EuMax := 6700.0, In_Raw := 4002, Percent := 0.012499999, PV := 0.8375);
   PT_802D : CM_AI_SCL := (RawMin := 4000, RawMax := 20000, EuMax := 6700.0, In_Raw := 3996, Percent := -0.024999999, PV := -1.675);
   PT_803 : CM_AI_SCL := (RawMin := 4000, RawMax := 20000, EuMax := 150.0, In_Raw := 4933, Percent := 5.8312497, PV := 8.746875);
   PT_806 : CM_AI_SCL := (RawMin := 4000, RawMax := 20000, EuMax := 3000.0, In_Raw := 4080, Percent := 0.5, PV := 15.0);
   PT_902 : CM_AI_SCL := (RawMin := 4000, RawMax := 20000, EuMax := 6700.0, In_Raw := 9719, Percent := 35.74375, PV := 2394.8313);
   Pull_Hold : BOOL;
   PUMP_CALC_FLOW : REAL;
   PUMP_CAVIT_PRESSURE_MARGIN : REAL := 500.0;   // HOW MUCH LOWER PUMP PT CAN BE THAN PT-902
   PUMP_CAVIT_PRESSURE_SP : REAL := 1894.8313;
   PWHMI_AtomizingStatus_OSR_OB : BOOL;
   PWHMI_AtomizingStatus_OSR_SB : BOOL;
   PWHMI_AtomizingStatusVerified : BOOL;
   PWHMI_BackfillStatus : BOOL;   // PWHMI Atomizer(s) Backfilling
   PWHMI_IdleStatus : BOOL;   // **future use
   PWHMI_MeltingStatus : BOOL;   // **future use
   PWHMI_OutletValveStatus : BOOL;
   PWHMI_Post_Atomize_TMR : TIMER := (PRE := 900000, ACC := 900000, EN := 1, DN := 1);
   PWHMI_Post_Collection_TMR : TIMER := (PRE := 900000, ACC := 900000, EN := 1, DN := 1);
   PWHMI_StartAtomizing : TIMER := (PRE := 2000);
   RCP_1000_COMMLOSS : BOOL;
   RCP_100_COMMLOSS : BOOL;
   RCP_600_COMMLOSS : BOOL;
   RCP_800_COMMLOSS : BOOL;
   REQUEST_ARGON_FROM_TK1100A : BOOL := 1;
   REQUEST_ARGON_FROM_TK700 : BOOL;
   Return_Stop_N2 : BOOL;
   Return_Stop_O2 : BOOL;
   SCR_1250 : BOOL;   // HXR-1250 SCR Active Signal
   SEND_AT2_PLANT_NOTICE : BOOL := 1;
   SEND_AT3_PLANT_NOTICE : BOOL := 1;
   SEND_PILOT_PLANT_NOTICE : BOOL := 1;
   START_ATOMIZE_DURING_PUMPUP : BOOL;
   SV_1000 : CM_DO_GENERIC;
   SV_1000B : CM_DO_GENERIC;
   SV_1000C : CM_DO_GENERIC := (EnergizeReq := 1);
   SV_1000D : CM_DO_GENERIC;
   SV_1000E : CM_DO_GENERIC := (Out := 1);
   SV_1001F : CM_DO_GENERIC := (Auto := 1, EnergizeReq := 1, Out := 1);
   SV_1002F : CM_DO_GENERIC := (EnergizeReq := 1, Out := 1);
   SV_1005_SPH : INT := 2600;
   SV_1005_SPL : INT := 2500;
   SV_1005X : CM_DO_GENERIC;
   SV_101AF : CM_DO_GENERIC := (Auto := 1, EnergizeReq := 1, Out := 1);
   SV_101AN : CM_DO_GENERIC := (Out := 1);
   SV_101AP : CM_DO_GENERIC := (FailPos := 1, Out := 1);
   SV_101BF : CM_DO_GENERIC := (Auto := 1, EnergizeReq := 1, Out := 1);
   SV_101BN : CM_DO_GENERIC := (Auto := 1);
   SV_101BP : CM_DO_GENERIC := (FailPos := 1, Auto := 1);
   SV_101BX : CM_DO_GENERIC;
   SV_101CF : CM_DO_GENERIC := (Auto := 1, EnergizeReq := 1, Out := 1);
   SV_101CN : CM_DO_GENERIC := (Auto := 1);
   SV_101CP : CM_DO_GENERIC := (FailPos := 1, Auto := 1);
   SV_101CX : CM_DO_GENERIC := (ILW := 1, EnergizeReq := 1);
   SV_102AF : CM_DO_GENERIC := (Auto := 1, EnergizeReq := 1, Out := 1);
   SV_102BF : CM_DO_GENERIC := (Auto := 1, EnergizeReq := 1, Out := 1);
   SV_102CF : CM_DO_GENERIC := (Auto := 1, EnergizeReq := 1, Out := 1);
   SV_1100P : CM_DO_GENERIC;
   SV_1104A : CM_DO_GENERIC;
   SV_1109AX : CM_DO_GENERIC;
   SV_1204 : CM_DO_GENERIC := (Out := 1);
   SV_1206 : CM_DO_GENERIC;
   SV_1207X : CM_DO_GENERIC := (Auto := 1);
   SV_1208X : CM_DO_GENERIC;
   SV_1221F : CM_DO_GENERIC := (Out := 1);
   SV_1251F : CM_DO_GENERIC := (Out := 1);
   SV_1276 : CM_DO_GENERIC;
   SV_1304A : CM_DO_GENERIC := (Auto := 1);
   SV_1304B : CM_DO_GENERIC := (Auto := 1);
   SV_1309AX : CM_DO_GENERIC := (Auto := 1);
   SV_1309BX : CM_DO_GENERIC := (Auto := 1);
   SV_200A : CM_DO_GENERIC;
   SV_200B : CM_DO_GENERIC;
   SV_202F : CM_DO_GENERIC := (Auto := 1, EnergizeReq := 1, Out := 1);
   SV_204F : CM_DO_GENERIC := (Auto := 1, EnergizeReq := 1, Out := 1);
   SV_205 : CM_DO_GENERIC := (Auto := 1);
   SV_205_ATOMIZE_OFFSET_SPH : REAL := 0.2;
   SV_205_ATOMIZE_OFFSET_SPL : REAL := 0.3;
   SV_205_FIXED : BOOL := 1;
   SV_205_IDLE_OFFSET_SPH : REAL := 0.2;
   SV_205_IDLE_OFFSET_SPL : REAL := 0.4;
   SV_205_Pressure_SPH : REAL := 1.4;
   SV_205_Pressure_SPH_TEST : REAL := 1.4;
   SV_205_Pressure_SPL : REAL := 1.2;
   SV_205_Pressure_SPL_TEST : REAL := 1.2;
   SV_206 : CM_DO_GENERIC := (Out := 1);
   SV_207F : CM_DO_GENERIC := (DeenergizeONS := 1);
   SV_221X : CM_DO_GENERIC := (Auto := 1);
   SV_221X_ONS : BOOL;
   SV_504F : CM_DO_GENERIC := (EnergizeReq := 1, Out := 1);
   SV_505X : CM_DO_GENERIC := (Auto := 1);
   SV_602A : CM_DO_GENERIC := (Out := 1);
   SV_603F : CM_DO_GENERIC := (EnergizeReq := 1, Out := 1);
   SV_605F : CM_DO_GENERIC := (Auto := 1, EnergizeReq := 1, Out := 1);
   SV_623X : CM_DO_GENERIC;
   SV_703X : CM_DO_GENERIC;
   SV_721AX : CM_DO_GENERIC;
   SV_721BX : CM_DO_GENERIC;
   SV_753F : CM_DO_GENERIC := (EnergizeReq := 1, Out := 1);
   SV_754F : CM_DO_GENERIC := (EnergizeReq := 1, Out := 1);
   SV_755F : CM_DO_GENERIC := (Auto := 1, DeenergizeONS := 1);
   SV_802AX : CM_DO_GENERIC := (Out := 1);
   SV_802AX_ONS : BOOL;
   SV_802BX : CM_DO_GENERIC := (Out := 1);
   SV_802BX_ONS : BOOL;
   SV_802CX : CM_DO_GENERIC := (Out := 1);
   SV_802CX_ONS : BOOL;
   SV_802DX : CM_DO_GENERIC := (Out := 1);
   SV_802DX_ONS : BOOL;
   TE_1003 : CM_AI_SCL := (RawMin := -4500, RawMax := 10000, EuMin := -450.0, EuMax := 1000.0, In_Raw := 531, Percent := 5.3100004, PV := 53.100006);
   TE_101A : CM_AI_SCL := (RawMin := -4500, RawMax := 10000, EuMin := -450.0, EuMax := 1000.0, In_Raw := 621, Percent := 6.2099977, PV := 62.099976);
   TE_101B : CM_AI_SCL := (RawMin := -4500, RawMax := 10000, EuMin := -450.0, EuMax := 1000.0, In_Raw := 677, Percent := 6.7700014, PV := 67.70001);
   TE_101C : CM_AI_SCL := (RawMin := -4500, RawMax := 10000, EuMin := -450.0, EuMax := 1000.0, In_Raw := 672, Percent := 6.720001, PV := 67.20001);
   TE_1201 : CM_AI_SCL := (RawMin := -4500, RawMax := 10000, EuMin := -450.0, EuMax := 1000.0, In_Raw := 554, Percent := 5.5399995, PV := 55.399994);
   TE_1202 : CM_AI_SCL := (RawMin := -4500, RawMax := 10000, EuMin := -450.0, EuMax := 1000.0, In_Raw := 547, Percent := 5.470001, PV := 54.700012);
   TE_1203 : CM_AI_SCL := (RawMin := -4500, RawMax := 10000, EuMin := -450.0, EuMax := 1000.0, In_Raw := 544, Percent := 5.439999, PV := 54.399994);
   TE_1204 : CM_AI_SCL := (RawMin := -4500, RawMax := 10000, EuMin := -450.0, EuMax := 1000.0, In_Raw := 549, Percent := 5.4899993, PV := 54.899994);
   TE_1205 : CM_AI_SCL := (RawMin := -4500, RawMax := 10000, EuMin := -450.0, EuMax := 1000.0, In_Raw := 555, Percent := 5.55, PV := 55.5);
   TE_1206 : CM_AI_SCL := (RawMin := -4500, RawMax := 10000, EuMin := -450.0, EuMax := 1000.0, In_Raw := 552, Percent := 5.520001, PV := 55.200012);
